// TwinCAT 3 PLC project SRC
// ProgramVersion: 3.1.4023.0
// libraries:
//   Tc2_Standard, * (Beckhoff Automation GmbH)
//   Tc2_System, * (Beckhoff Automation GmbH)
//   Tc3_JsonXml, * (Beckhoff Automation GmbH)
//   Tc3_Module, * (Beckhoff Automation GmbH)
// project tree:
//   DUTs/ENUM/ eCellState.TcDUT, eState.TcDUT
//   DUTs/STRUCT/HandledIO/Inputs/ st_IO_Inputs.TcDUT, st_PressureTransducer_Input.TcDUT, st_Robot_Input.TcDUT
//   DUTs/STRUCT/HandledIO/Outputs/ st_IO_Outputs.TcDUT, st_Pump_Output.TcDUT, st_Robot_Output.TcDUT
//   DUTs/STRUCT/Config/ ST_Configuration.TcDUT
//   DUTs/STRUCT/HMI/inputs/ st_PLCtoHMI_VariantControl.TcDUT, st_PLCtoHMI.TcDUT, st_PLCtoHMI_Hydrualics.TcDUT, st_PLCtoHMI_Cell.TcDUT, st_PLCtoHMI_PressureTrans.TcDUT, st_PLCtoHMI_Pump.TcDUT, st_PLCtoHMI_Robot.TcDUT
//   DUTs/STRUCT/HMI/outputs/ st_HMItoPLC.TcDUT, st_HMItoPLC_Cell.TcDUT, st_HMItoPLC_HMI.TcDUT, st_HMItoPLC_VariantControl.TcDUT
//   DUTs/STRUCT/IO/Base/ EtcMasterBase_62654B43.TcDUT, EtcSlaveBase_82538BE2.TcDUT, EtcSlaveBoxBase_77A0E4A7.TcDUT, EtcSlaveEndTerminalBase_866C7F0C.TcDUT, EtcSlaveTerminalBase_947E5A46.TcDUT, InputBase_8311D824.TcDUT, OutputBase_10CEE7DE.TcDUT, SyncUnitsBase_AD6C35CE.TcDUT, SyncUnitTaskBase_FCD3CBF3.TcDUT, SyncUnitTasksBase_7C8711EB.TcDUT
//   DUTs/STRUCT/IO/Boxes/ EK1100_1FC0878B.TcDUT, EL2634_7B64371E.TcDUT, EL3024_C4269E32.TcDUT, KRC4_secondary_EL6695_4F43E7C3.TcDUT
//   DUTs/STRUCT/IO/Devices/ SyncUnits_67D36DDA.TcDUT, SyncUnitTasks_4BE01469.TcDUT, SyncUnitTask_AB2F5079.TcDUT
//   DUTs/STRUCT/IO/PdoEntries/ FSOE_8292E3BB.TcDUT, FSOE_892AE692.TcDUT, Status_F2CE6D91.TcDUT
//   DUTs/STRUCT/IO/PDOs/ AI_Standard_Channel_4A394481.TcDUT, Channel_42CA91F7.TcDUT, Compact_1DE69B90.TcDUT, InfoData_32EB74EA.TcDUT, InfoData_6F19DB2B.TcDUT, InfoData_8649EEEB.TcDUT, InfoData_90184F0C.TcDUT, InfoData_E68C61CD.TcDUT, Inputs_A65FACA4.TcDUT, Inputs_Bitf_43DA21F5.TcDUT, Module_1_Sync_Inputs_26A07CFD.TcDUT, Module_2_Safety_Data_Bitf_8_Byte_x_D7FC8792.TcDUT, Module_3_Default_IO_1C907BA3.TcDUT, Outputs_23C0ED1D.TcDUT, Outputs_Bitf_2744F336.TcDUT, Std_In_4_Bytes_89628F68.TcDUT, Std_Out_4_Bytes_1F5BD6B7.TcDUT, WcState_0B2B16F9.TcDUT, WcState_9091E0EB.TcDUT
//   DUTs/STRUCT/IO/Topology/ E_Bus_F0495AE1.TcDUT, Term_1_EK1100_53501D32.TcDUT
//   / PlcTask.TcTTO
//   POUs/Cell/BaseClasses/ StateMachineBase.TcPOU
//   POUs/Cell/ FB_Cell.TcPOU
//   POUs/Cell/Hardware_IO/ FB_Topology.TcPOU
//   POUs/Cell/Hydrualics/ FB_HydrualicSystem.TcPOU
//   POUs/Cell/Hydrualics/PressureSensor/ FB_PressureSensor.TcPOU
//   POUs/Cell/Hydrualics/PressureSensor/Types/ FB_GenericBrand_Transceiver.TcPOU, FB_PressureTransceiver_Sim.TcPOU
//   POUs/Cell/Hydrualics/Pump/ FB_Pump.TcPOU
//   POUs/Cell/Hydrualics/Pump/Types/ FB_Pump_HPU.TcPOU, FB_Pump_RelayOnly.TcPOU, FB_Pump_Simulator.TcPOU
//   POUs/Cell/Robots/6_axis/Types/ FB_Fanuc.TcPOU, FB_Kuka_KRC2.TcPOU, FB_Kuka_KRC4.TcPOU, FB_Robot_Simulator.TcPOU
//   POUs/Cell/Robots/ FB_Robot.TcPOU
//   POUs/Cell/Robots/Gantry/Types/ FB_SomeGrantryRobot.TcPOU
//   POUs/Cell/_Interface/ I_HydrualicPump.TcIO, I_PressureSensor.TcIO, I_Robot.TcIO
//   POUs/ FB_VariantControl.TcPOU, MAIN.TcPOU
//   POUs/Functions/ Queue_FIFO.TcPOU, Scale.TcPOU
//   POUs/HMI/ FB_HMI.TcPOU
//   GVLs/ GVL_iXlinker.TcGVL

CONFIGURATION SRC
    RESOURCE PLC ON TwinCAT3
        TASK PlcTask(INTERVAL := T#10ms, PRIORITY := 20);
        PROGRAM MAIN WITH PlcTask : MAIN;
    END_RESOURCE
END_CONFIGURATION

// ---- DUTs/ENUM/eCellState.TcDUT
TYPE eCellState :
(
	eCellState_Manual, eCellState_Automatic, eCellState_Error
);
END_TYPE

// ---- DUTs/ENUM/eState.TcDUT
{attribute 'strict'}
{attribute 'to_string'}
TYPE eState :
(
	eState_Idle, eState_Startup, eState_Ready, eState_Running, eState_Complete, eState_Holding,
	eState_Held, eState_Stopping, eState_Stopped, eState_Error, eState_Independent, eState_Resetting, eState_Restarting,
	eState_Warmup
);
END_TYPE

// ---- DUTs/STRUCT/HandledIO/Inputs/st_IO_Inputs.TcDUT
TYPE st_IO_Inputs :
STRUCT
    robot :ST_Robot_Input;
    pressureTransducer : ST_PressureTransducer_Input;
END_STRUCT
END_TYPE

// ---- DUTs/STRUCT/HandledIO/Inputs/st_PressureTransducer_Input.TcDUT
TYPE st_PressureTransducer_Input :
STRUCT
	value : LREAL;
END_STRUCT
END_TYPE

// ---- DUTs/STRUCT/HandledIO/Inputs/st_Robot_Input.TcDUT
TYPE st_Robot_Input :
STRUCT
    fault : BOOL;
END_STRUCT
END_TYPE

// ---- DUTs/STRUCT/HandledIO/Outputs/st_IO_Outputs.TcDUT
TYPE st_IO_Outputs :
STRUCT
    hydroPump : ST_Pump_Output;
    robot : ST_Robot_Output;
END_STRUCT
END_TYPE

// ---- DUTs/STRUCT/HandledIO/Outputs/st_Pump_Output.TcDUT
TYPE st_Pump_Output :
STRUCT
	On : BOOL;
END_STRUCT
END_TYPE

// ---- DUTs/STRUCT/HandledIO/Outputs/st_Robot_Output.TcDUT
TYPE st_Robot_Output :
STRUCT
    fault : BOOL;
END_STRUCT
END_TYPE

// ---- DUTs/STRUCT/Config/ST_Configuration.TcDUT
TYPE ST_Configuration :
STRUCT
	sVersionHW : STRING;
	sVersionSW : STRING;

	// Which variant is active
	bIsV1_0_0 		: BOOL;
	bIsSimulator 	: BOOL;

	// Hydrualic pump definition
	bHasPump : BOOL;
	sPumpType : STRING;
	
	// Pressure sensor definition
	bHasPressureSensor : BOOL;
	sPressureSensorType : STRING;
    
    // Robot definition
    bHasRobot : BOOL;
    sRobotType : STRING;
END_STRUCT
END_TYPE

// ---- DUTs/STRUCT/HMI/inputs/st_PLCtoHMI_VariantControl.TcDUT
TYPE st_PLCtoHMI_VariantControl :
STRUCT
    bNeedsCellDefinition : BOOL;
END_STRUCT
END_TYPE

// ---- DUTs/STRUCT/HMI/inputs/st_PLCtoHMI.TcDUT
TYPE st_PLCtoHMI :
STRUCT
    cell : st_PLCtoHMI_Cell;
    robot : st_PLCtoHMI_Robot;
    hydrualics : st_PLCtoHMI_Hydrualics;
    variantControl : st_PLCtoHMI_VariantControl;
    //hmi : st_PLCtoHMI_HMI;
END_STRUCT
END_TYPE

// ---- DUTs/STRUCT/HMI/inputs/st_PLCtoHMI_Hydrualics.TcDUT
TYPE st_PLCtoHMI_Hydrualics :
STRUCT
    state : eState;
    psiSensor : st_PLCtoHMI_PressureTrans;
    pump : st_PLCtoHMI_Pump;
END_STRUCT
END_TYPE

// ---- DUTs/STRUCT/HMI/inputs/st_PLCtoHMI_Cell.TcDUT
TYPE st_PLCtoHMI_Cell :
STRUCT
    state : eCellState;
    bPower : BOOL; // power hydrualics maybe?
    bGoToManual: BOOL;
	bGoToAuto: BOOL;
	bReset : BOOL;
END_STRUCT
END_TYPE

// ---- DUTs/STRUCT/HMI/inputs/st_PLCtoHMI_PressureTrans.TcDUT
TYPE st_PLCtoHMI_PressureTrans :
STRUCT
    value : LREAL;
END_STRUCT
END_TYPE

// ---- DUTs/STRUCT/HMI/inputs/st_PLCtoHMI_Pump.TcDUT
TYPE st_PLCtoHMI_Pump :
STRUCT
    state : eState;
END_STRUCT
END_TYPE

// ---- DUTs/STRUCT/HMI/inputs/st_PLCtoHMI_Robot.TcDUT
TYPE st_PLCtoHMI_Robot :
STRUCT
    state : eState;
END_STRUCT
END_TYPE

// ---- DUTs/STRUCT/HMI/outputs/st_HMItoPLC.TcDUT
TYPE st_HMItoPLC :
STRUCT
    cell : st_HMItoPLC_Cell;
    hmi : st_HMItoPLC_HMI;
    variantControl : st_HMItoPLC_VariantControl;
END_STRUCT
END_TYPE

// ---- DUTs/STRUCT/HMI/outputs/st_HMItoPLC_Cell.TcDUT
TYPE st_HMItoPLC_Cell :
STRUCT
    bPower : BOOL; // power hydrualics maybe?
    bGoToManual: BOOL;
	bGoToAuto: BOOL;
	bReset : BOOL;
END_STRUCT
END_TYPE

// ---- DUTs/STRUCT/HMI/outputs/st_HMItoPLC_HMI.TcDUT
TYPE st_HMItoPLC_HMI :
STRUCT
    bAutoManual_btn : BOOL;
    bShowResetBtn : BOOL;
END_STRUCT
END_TYPE

// ---- DUTs/STRUCT/HMI/outputs/st_HMItoPLC_VariantControl.TcDUT
TYPE st_HMItoPLC_VariantControl :
STRUCT
    bExportJSON : BOOL;
    bWriteJSON : BOOL;
    Config : ST_Configuration;
    bNeedsCellDefinition : BOOL;
END_STRUCT
END_TYPE

// ---- DUTs/STRUCT/IO/Base/EtcMasterBase_62654B43.TcDUT

TYPE EtcMasterBase_62654B43 :
STRUCT
END_STRUCT
END_TYPE

// ---- DUTs/STRUCT/IO/Base/EtcSlaveBase_82538BE2.TcDUT

TYPE EtcSlaveBase_82538BE2 :
STRUCT
END_STRUCT
END_TYPE

// ---- DUTs/STRUCT/IO/Base/EtcSlaveBoxBase_77A0E4A7.TcDUT

{attribute clr[Container(Layout.Stack)]}
{attribute clr[Group(Layout.GroupBox)]}
{attribute addProperty PreviousPort "Unknown"}
{attribute addProperty SyncUnit "Unknown"}
TYPE EtcSlaveBoxBase_77A0E4A7 EXTENDS EtcSlaveBase_82538BE2 :
STRUCT
END_STRUCT
END_TYPE

// ---- DUTs/STRUCT/IO/Base/EtcSlaveEndTerminalBase_866C7F0C.TcDUT

{attribute clr[Container(Layout.Stack)]}
{attribute clr[Group(Layout.GroupBox)]}
{attribute addProperty PreviousPort "Unknown"}
{attribute addProperty SyncUnit "Unknown"}
TYPE EtcSlaveEndTerminalBase_866C7F0C EXTENDS EtcSlaveBase_82538BE2 :
STRUCT
END_STRUCT
END_TYPE

// ---- DUTs/STRUCT/IO/Base/EtcSlaveTerminalBase_947E5A46.TcDUT

{attribute clr[Container(Layout.Stack)]}
{attribute clr[Group(Layout.GroupBox)]}
{attribute addProperty PreviousPort "Unknown"}
{attribute addProperty SyncUnit "Unknown"}
TYPE EtcSlaveTerminalBase_947E5A46 EXTENDS EtcSlaveBase_82538BE2 :
STRUCT
END_STRUCT
END_TYPE

// ---- DUTs/STRUCT/IO/Base/InputBase_8311D824.TcDUT

TYPE InputBase_8311D824 :
STRUCT
END_STRUCT
END_TYPE

// ---- DUTs/STRUCT/IO/Base/OutputBase_10CEE7DE.TcDUT

TYPE OutputBase_10CEE7DE :
STRUCT
END_STRUCT
END_TYPE

// ---- DUTs/STRUCT/IO/Base/SyncUnitsBase_AD6C35CE.TcDUT

TYPE SyncUnitsBase_AD6C35CE :
STRUCT
END_STRUCT
END_TYPE

// ---- DUTs/STRUCT/IO/Base/SyncUnitTaskBase_FCD3CBF3.TcDUT

TYPE SyncUnitTaskBase_FCD3CBF3 :
STRUCT
END_STRUCT
END_TYPE

// ---- DUTs/STRUCT/IO/Base/SyncUnitTasksBase_7C8711EB.TcDUT

TYPE SyncUnitTasksBase_7C8711EB :
STRUCT
END_STRUCT
END_TYPE

// ---- DUTs/STRUCT/IO/Boxes/EK1100_1FC0878B.TcDUT
{attribute 'GeneratedUsingTerminal: EK1100-0000-0018'}
{attribute addProperty VendorId "#x00000002"}
{attribute addProperty BoxType "EK1100-0000-0018"}
{attribute addProperty Description "EK1100 EtherCAT Coupler (2A E-Bus)"}
{attribute addProperty Physics "YKY"}
{attribute addProperty Id "InfoDataAT %I*InfoData_6F19DB2B2"}
{attribute addProperty CRC "532711307"}
{attribute addProperty Size "2"}
TYPE EK1100_1FC0878B EXTENDS EtcSlaveBoxBase_77A0E4A7 :
STRUCT
	{attribute addProperty Name "InfoData"}
	InfoData : InfoData_6F19DB2B;
END_STRUCT
END_TYPE

// ---- DUTs/STRUCT/IO/Boxes/EL2634_7B64371E.TcDUT
{attribute 'GeneratedUsingTerminal: EL2634-0000-0017'}
{attribute addProperty VendorId "#x00000002"}
{attribute addProperty BoxType "EL2634-0000-0017"}
{attribute addProperty Description "EL2634 4Ch. Relay Output, NO (250V AC / 30V DC)"}
{attribute addProperty Physics "KK"}
{attribute addProperty Id "Channel_1AT %Q*Channel_42CA91F71Channel_2AT %Q*Channel_42CA91F71Channel_3AT %Q*Channel_42CA91F71Channel_4AT %Q*Channel_42CA91F71WcStateAT %I*WcState_0B2B16F91InfoDataAT %I*InfoData_6F19DB2B2"}
{attribute addProperty CRC "2070165278"}
{attribute addProperty Size "7"}
TYPE EL2634_7B64371E EXTENDS EtcSlaveTerminalBase_947E5A46 :
STRUCT
	{attribute addProperty Name "Channel_1"}
	Channel_1 : Channel_42CA91F7;
	{attribute addProperty Name "Channel_2"}
	Channel_2 : Channel_42CA91F7;
	{attribute addProperty Name "Channel_3"}
	Channel_3 : Channel_42CA91F7;
	{attribute addProperty Name "Channel_4"}
	Channel_4 : Channel_42CA91F7;
	{attribute addProperty Name "WcState"}
	WcState : WcState_0B2B16F9;
	{attribute addProperty Name "InfoData"}
	InfoData : InfoData_6F19DB2B;
END_STRUCT
END_TYPE

// ---- DUTs/STRUCT/IO/Boxes/EL3024_C4269E32.TcDUT
{attribute 'GeneratedUsingTerminal: EL3024-0000-0019'}
{attribute addProperty VendorId "#x00000002"}
{attribute addProperty BoxType "EL3024-0000-0019"}
{attribute addProperty Description "EL3024 4Ch. Ana. Input 4-20mA DIFF"}
{attribute addProperty Physics "KK"}
{attribute addProperty Id "AI_Standard_Channel_1AT %I*AI_Standard_Channel_4A3944819AI_Standard_Channel_2AT %I*AI_Standard_Channel_4A3944819AI_Standard_Channel_3AT %I*AI_Standard_Channel_4A3944819AI_Standard_Channel_4AT %I*AI_Standard_Channel_4A3944819WcStateAT %I*WcState_9091E0EB2InfoDataAT %I*InfoData_32EB74EA10"}
{attribute addProperty CRC "3290865202"}
{attribute addProperty Size "48"}
TYPE EL3024_C4269E32 EXTENDS EtcSlaveTerminalBase_947E5A46 :
STRUCT
	{attribute addProperty Name "AI_Standard_Channel_1"}
	AI_Standard_Channel_1 : AI_Standard_Channel_4A394481;
	{attribute addProperty Name "AI_Standard_Channel_2"}
	AI_Standard_Channel_2 : AI_Standard_Channel_4A394481;
	{attribute addProperty Name "AI_Standard_Channel_3"}
	AI_Standard_Channel_3 : AI_Standard_Channel_4A394481;
	{attribute addProperty Name "AI_Standard_Channel_4"}
	AI_Standard_Channel_4 : AI_Standard_Channel_4A394481;
	{attribute addProperty Name "WcState"}
	WcState : WcState_9091E0EB;
	{attribute addProperty Name "InfoData"}
	InfoData : InfoData_32EB74EA;
END_STRUCT
END_TYPE

// ---- DUTs/STRUCT/IO/Boxes/KRC4_secondary_EL6695_4F43E7C3.TcDUT
{attribute 'GeneratedUsingTerminal: KRC4 secondary EL6695-1001-0004'}
{attribute addProperty VendorId "#x000060c8"}
{attribute addProperty BoxType "KRC4 secondary EL6695-1001-0004"}
{attribute addProperty Description "KRC4 secondary EL6695-1001"}
{attribute addProperty Physics "YY"}
{attribute addProperty Id "Module_1_Sync_InputsModule_1_Sync_Inputs_26A07CFD3Module_2_Safety_Data_Bitf_8_Byte_xModule_2_Safety_Data_Bitf_8_Byte_x_D7FC8792150Module_3_Default_IOModule_3_Default_IO_1C907BA38WcStateAT %I*WcState_9091E0EB2InfoDataAT %I*InfoData_90184F0C16"}
{attribute addProperty CRC "1329850307"}
{attribute addProperty Size "179"}
TYPE KRC4_secondary_EL6695_4F43E7C3 EXTENDS EtcSlaveBoxBase_77A0E4A7 :
STRUCT
	{attribute addProperty Name "Module_1_Sync_Inputs"}
	Module_1_Sync_Inputs : Module_1_Sync_Inputs_26A07CFD;
	{attribute addProperty Name "Module_2_Safety_Data_Bitf_8_Byte_x"}
	Module_2_Safety_Data_Bitf_8_Byte_x : Module_2_Safety_Data_Bitf_8_Byte_x_D7FC8792;
	{attribute addProperty Name "Module_3_Default_IO"}
	Module_3_Default_IO : Module_3_Default_IO_1C907BA3;
	{attribute addProperty Name "WcState"}
	WcState : WcState_9091E0EB;
	{attribute addProperty Name "InfoData"}
	InfoData : InfoData_90184F0C;
END_STRUCT
END_TYPE

// ---- DUTs/STRUCT/IO/Devices/SyncUnits_67D36DDA.TcDUT
{attribute 'GeneratedUsingTerminal: '}
{attribute addProperty BoxType ""}
{attribute addProperty Id "_defaultAT %I*SyncUnitTasks_4BE0146918"}
{attribute addProperty CRC "1741909466"}
{attribute addProperty Size "18"}
TYPE SyncUnits_67D36DDA EXTENDS SyncUnitsBase_AD6C35CE :
STRUCT
	{attribute addProperty Name "_default"}
	_default : SyncUnitTasks_4BE01469;
END_STRUCT
END_TYPE

// ---- DUTs/STRUCT/IO/Devices/SyncUnitTasks_4BE01469.TcDUT
{attribute 'GeneratedUsingTerminal: '}
{attribute addProperty BoxType ""}
{attribute addProperty Id "unreferencedAT %I*SyncUnitTask_AB2F50799PlcTaskAT %I*SyncUnitTask_AB2F50799"}
{attribute addProperty CRC "1272976489"}
{attribute addProperty Size "18"}
TYPE SyncUnitTasks_4BE01469 EXTENDS SyncUnitTasksBase_7C8711EB :
STRUCT
	{attribute addProperty Name "unreferenced"}
	unreferenced : SyncUnitTask_AB2F5079;
	{attribute addProperty Name "PlcTask"}
	PlcTask : SyncUnitTask_AB2F5079;
END_STRUCT
END_TYPE

// ---- DUTs/STRUCT/IO/Devices/SyncUnitTask_AB2F5079.TcDUT
{attribute 'GeneratedUsingTerminal: IODEVICETYPE_ETHERCATPROT'}
{attribute addProperty BoxType "IODEVICETYPE_ETHERCATPROT"}
{attribute addProperty Id "WcStateAT %I*WcState_0B2B16F91InfoDataAT %I*InfoData_8649EEEB8"}
{attribute addProperty CRC "2872004729"}
{attribute addProperty Size "9"}
TYPE SyncUnitTask_AB2F5079 EXTENDS SyncUnitTaskBase_FCD3CBF3 :
STRUCT
	{attribute addProperty Name "WcState"}
	WcState : WcState_0B2B16F9;
	{attribute addProperty Name "InfoData"}
	InfoData : InfoData_8649EEEB;
END_STRUCT
END_TYPE

// ---- DUTs/STRUCT/IO/PdoEntries/FSOE_8292E3BB.TcDUT
{attribute 'GeneratedUsingTerminal: KRC4 secondary EL6695-1001-0004'}
{attribute addProperty BoxType "KRC4 secondary EL6695-1001-0004"}
{attribute addProperty Id "FSOE_CommandUSINT1FSOE_Out_D_0_RES_1BOOL1FSOE_Out_D_0_NHEBOOL1FSOE_Out_D_0_BSBOOL1FSOE_Out_D_0_QBSBOOL1FSOE_Out_D_0_SHS1BOOL1FSOE_Out_D_0_SHS2BOOL1FSOE_Out_D_0_E2BOOL1FSOE_Out_D_0_E7BOOL1FSOE_Out_D_0_US2BOOL1FSOE_Out_D_0_SBHBOOL1FSOE_Out_D_0_RES_4BOOL1FSOE_Out_D_0_RES_5BOOL1FSOE_Out_D_0_RES_6BOOL1FSOE_Out_D_0_RES_7BOOL1FSOE_Out_D_0_RES_8BOOL1FSOE_Out_D_0_SPABOOL1FSOE_Master_CRC_0UINT2FSOE_Out_D_1_JRBOOL1FSOE_Out_D_1_VREDBOOL1FSOE_Out_D_1_SBH_1BOOL1FSOE_Out_D_1_SBH_2BOOL1FSOE_Out_D_1_SBH_3BOOL1FSOE_Out_D_1_SBH_4BOOL1FSOE_Out_D_1_SBH_5BOOL1FSOE_Out_D_1_SBH_6BOOL1FSOE_Out_D_1_RES_1BOOL1FSOE_Out_D_1_RES_2BOOL1FSOE_Out_D_1_RES_3BOOL1FSOE_Out_D_1_RES_4BOOL1FSOE_Out_D_1_RES_5BOOL1FSOE_Out_D_1_RES_6BOOL1FSOE_Out_D_1_RES_7BOOL1FSOE_Out_D_1_RES_8BOOL1FSOE_Master_CRC_1UINT2FSOE_Out_D_2_UER1BOOL1FSOE_Out_D_2_UER2BOOL1FSOE_Out_D_2_UER3BOOL1FSOE_Out_D_2_UER4BOOL1FSOE_Out_D_2_UER5BOOL1FSOE_Out_D_2_UER6BOOL1FSOE_Out_D_2_UER7BOOL1FSOE_Out_D_2_UER8BOOL1FSOE_Out_D_2_UER9BOOL1FSOE_Out_D_2_UER10BOOL1FSOE_Out_D_2_UER11BOOL1FSOE_Out_D_2_UER12BOOL1FSOE_Out_D_2_UER13BOOL1FSOE_Out_D_2_UER14BOOL1FSOE_Out_D_2_UER15BOOL1FSOE_Out_D_2_UER16BOOL1FSOE_Master_CRC_2UINT2FSOE_Out_D_3_WZ1BOOL1FSOE_Out_D_3_WZ2BOOL1FSOE_Out_D_3_WZ3BOOL1FSOE_Out_D_3_WZ4BOOL1FSOE_Out_D_3_WZ5BOOL1FSOE_Out_D_3_WZ6BOOL1FSOE_Out_D_3_WZ7BOOL1FSOE_Out_D_3_WZ8BOOL1FSOE_Out_D_3_WZ9BOOL1FSOE_Out_D_3_WZ10BOOL1FSOE_Out_D_3_WZ11BOOL1FSOE_Out_D_3_WZ12BOOL1FSOE_Out_D_3_WZ13BOOL1FSOE_Out_D_3_WZ14BOOL1FSOE_Out_D_3_WZ15BOOL1FSOE_Out_D_3_WZ16BOOL1FSOE_Master_CRC_3UINT2FSOE_ConnIDUINT2"}
{attribute addProperty CRC "2190664635"}
{attribute addProperty Size "75"}
TYPE FSOE_8292E3BB :
STRUCT
	{attribute addProperty Name "FSOE_Command"}
	FSOE_Command : USINT;
	{attribute addProperty Name "FSOE_Out_D_0_RES_1"}
	FSOE_Out_D_0_RES_1 : BOOL;
	{attribute addProperty Name "FSOE_Out_D_0_NHE"}
	FSOE_Out_D_0_NHE : BOOL;
	{attribute addProperty Name "FSOE_Out_D_0_BS"}
	FSOE_Out_D_0_BS : BOOL;
	{attribute addProperty Name "FSOE_Out_D_0_QBS"}
	FSOE_Out_D_0_QBS : BOOL;
	{attribute addProperty Name "FSOE_Out_D_0_SHS1"}
	FSOE_Out_D_0_SHS1 : BOOL;
	{attribute addProperty Name "FSOE_Out_D_0_SHS2"}
	FSOE_Out_D_0_SHS2 : BOOL;
	{attribute addProperty Name "FSOE_Out_D_0_E2"}
	FSOE_Out_D_0_E2 : BOOL;
	{attribute addProperty Name "FSOE_Out_D_0_E7"}
	FSOE_Out_D_0_E7 : BOOL;
	{attribute addProperty Name "FSOE_Out_D_0_US2"}
	FSOE_Out_D_0_US2 : BOOL;
	{attribute addProperty Name "FSOE_Out_D_0_SBH"}
	FSOE_Out_D_0_SBH : BOOL;
	{attribute addProperty Name "FSOE_Out_D_0_RES_4"}
	FSOE_Out_D_0_RES_4 : BOOL;
	{attribute addProperty Name "FSOE_Out_D_0_RES_5"}
	FSOE_Out_D_0_RES_5 : BOOL;
	{attribute addProperty Name "FSOE_Out_D_0_RES_6"}
	FSOE_Out_D_0_RES_6 : BOOL;
	{attribute addProperty Name "FSOE_Out_D_0_RES_7"}
	FSOE_Out_D_0_RES_7 : BOOL;
	{attribute addProperty Name "FSOE_Out_D_0_RES_8"}
	FSOE_Out_D_0_RES_8 : BOOL;
	{attribute addProperty Name "FSOE_Out_D_0_SPA"}
	FSOE_Out_D_0_SPA : BOOL;
	{attribute addProperty Name "FSOE_Master_CRC_0"}
	FSOE_Master_CRC_0 : UINT;
	{attribute addProperty Name "FSOE_Out_D_1_JR"}
	FSOE_Out_D_1_JR : BOOL;
	{attribute addProperty Name "FSOE_Out_D_1_VRED"}
	FSOE_Out_D_1_VRED : BOOL;
	{attribute addProperty Name "FSOE_Out_D_1_SBH_1"}
	FSOE_Out_D_1_SBH_1 : BOOL;
	{attribute addProperty Name "FSOE_Out_D_1_SBH_2"}
	FSOE_Out_D_1_SBH_2 : BOOL;
	{attribute addProperty Name "FSOE_Out_D_1_SBH_3"}
	FSOE_Out_D_1_SBH_3 : BOOL;
	{attribute addProperty Name "FSOE_Out_D_1_SBH_4"}
	FSOE_Out_D_1_SBH_4 : BOOL;
	{attribute addProperty Name "FSOE_Out_D_1_SBH_5"}
	FSOE_Out_D_1_SBH_5 : BOOL;
	{attribute addProperty Name "FSOE_Out_D_1_SBH_6"}
	FSOE_Out_D_1_SBH_6 : BOOL;
	{attribute addProperty Name "FSOE_Out_D_1_RES_1"}
	FSOE_Out_D_1_RES_1 : BOOL;
	{attribute addProperty Name "FSOE_Out_D_1_RES_2"}
	FSOE_Out_D_1_RES_2 : BOOL;
	{attribute addProperty Name "FSOE_Out_D_1_RES_3"}
	FSOE_Out_D_1_RES_3 : BOOL;
	{attribute addProperty Name "FSOE_Out_D_1_RES_4"}
	FSOE_Out_D_1_RES_4 : BOOL;
	{attribute addProperty Name "FSOE_Out_D_1_RES_5"}
	FSOE_Out_D_1_RES_5 : BOOL;
	{attribute addProperty Name "FSOE_Out_D_1_RES_6"}
	FSOE_Out_D_1_RES_6 : BOOL;
	{attribute addProperty Name "FSOE_Out_D_1_RES_7"}
	FSOE_Out_D_1_RES_7 : BOOL;
	{attribute addProperty Name "FSOE_Out_D_1_RES_8"}
	FSOE_Out_D_1_RES_8 : BOOL;
	{attribute addProperty Name "FSOE_Master_CRC_1"}
	FSOE_Master_CRC_1 : UINT;
	{attribute addProperty Name "FSOE_Out_D_2_UER1"}
	FSOE_Out_D_2_UER1 : BOOL;
	{attribute addProperty Name "FSOE_Out_D_2_UER2"}
	FSOE_Out_D_2_UER2 : BOOL;
	{attribute addProperty Name "FSOE_Out_D_2_UER3"}
	FSOE_Out_D_2_UER3 : BOOL;
	{attribute addProperty Name "FSOE_Out_D_2_UER4"}
	FSOE_Out_D_2_UER4 : BOOL;
	{attribute addProperty Name "FSOE_Out_D_2_UER5"}
	FSOE_Out_D_2_UER5 : BOOL;
	{attribute addProperty Name "FSOE_Out_D_2_UER6"}
	FSOE_Out_D_2_UER6 : BOOL;
	{attribute addProperty Name "FSOE_Out_D_2_UER7"}
	FSOE_Out_D_2_UER7 : BOOL;
	{attribute addProperty Name "FSOE_Out_D_2_UER8"}
	FSOE_Out_D_2_UER8 : BOOL;
	{attribute addProperty Name "FSOE_Out_D_2_UER9"}
	FSOE_Out_D_2_UER9 : BOOL;
	{attribute addProperty Name "FSOE_Out_D_2_UER10"}
	FSOE_Out_D_2_UER10 : BOOL;
	{attribute addProperty Name "FSOE_Out_D_2_UER11"}
	FSOE_Out_D_2_UER11 : BOOL;
	{attribute addProperty Name "FSOE_Out_D_2_UER12"}
	FSOE_Out_D_2_UER12 : BOOL;
	{attribute addProperty Name "FSOE_Out_D_2_UER13"}
	FSOE_Out_D_2_UER13 : BOOL;
	{attribute addProperty Name "FSOE_Out_D_2_UER14"}
	FSOE_Out_D_2_UER14 : BOOL;
	{attribute addProperty Name "FSOE_Out_D_2_UER15"}
	FSOE_Out_D_2_UER15 : BOOL;
	{attribute addProperty Name "FSOE_Out_D_2_UER16"}
	FSOE_Out_D_2_UER16 : BOOL;
	{attribute addProperty Name "FSOE_Master_CRC_2"}
	FSOE_Master_CRC_2 : UINT;
	{attribute addProperty Name "FSOE_Out_D_3_WZ1"}
	FSOE_Out_D_3_WZ1 : BOOL;
	{attribute addProperty Name "FSOE_Out_D_3_WZ2"}
	FSOE_Out_D_3_WZ2 : BOOL;
	{attribute addProperty Name "FSOE_Out_D_3_WZ3"}
	FSOE_Out_D_3_WZ3 : BOOL;
	{attribute addProperty Name "FSOE_Out_D_3_WZ4"}
	FSOE_Out_D_3_WZ4 : BOOL;
	{attribute addProperty Name "FSOE_Out_D_3_WZ5"}
	FSOE_Out_D_3_WZ5 : BOOL;
	{attribute addProperty Name "FSOE_Out_D_3_WZ6"}
	FSOE_Out_D_3_WZ6 : BOOL;
	{attribute addProperty Name "FSOE_Out_D_3_WZ7"}
	FSOE_Out_D_3_WZ7 : BOOL;
	{attribute addProperty Name "FSOE_Out_D_3_WZ8"}
	FSOE_Out_D_3_WZ8 : BOOL;
	{attribute addProperty Name "FSOE_Out_D_3_WZ9"}
	FSOE_Out_D_3_WZ9 : BOOL;
	{attribute addProperty Name "FSOE_Out_D_3_WZ10"}
	FSOE_Out_D_3_WZ10 : BOOL;
	{attribute addProperty Name "FSOE_Out_D_3_WZ11"}
	FSOE_Out_D_3_WZ11 : BOOL;
	{attribute addProperty Name "FSOE_Out_D_3_WZ12"}
	FSOE_Out_D_3_WZ12 : BOOL;
	{attribute addProperty Name "FSOE_Out_D_3_WZ13"}
	FSOE_Out_D_3_WZ13 : BOOL;
	{attribute addProperty Name "FSOE_Out_D_3_WZ14"}
	FSOE_Out_D_3_WZ14 : BOOL;
	{attribute addProperty Name "FSOE_Out_D_3_WZ15"}
	FSOE_Out_D_3_WZ15 : BOOL;
	{attribute addProperty Name "FSOE_Out_D_3_WZ16"}
	FSOE_Out_D_3_WZ16 : BOOL;
	{attribute addProperty Name "FSOE_Master_CRC_3"}
	FSOE_Master_CRC_3 : UINT;
	{attribute addProperty Name "FSOE_ConnID"}
	FSOE_ConnID : UINT;
END_STRUCT
END_TYPE

// ---- DUTs/STRUCT/IO/PdoEntries/FSOE_892AE692.TcDUT
{attribute 'GeneratedUsingTerminal: KRC4 secondary EL6695-1001-0004'}
{attribute addProperty BoxType "KRC4 secondary EL6695-1001-0004"}
{attribute addProperty Id "FSOE_CommandUSINT1FSOE_Inp_D_0_NHLBOOL1FSOE_Inp_D_0_AFBOOL1FSOE_Inp_D_0_FFBOOL1FSOE_Inp_D_0_ZSBOOL1FSOE_Inp_D_0_PEBOOL1FSOE_Inp_D_0_EXTBOOL1FSOE_Inp_D_0_T1BOOL1FSOE_Inp_D_0_T2BOOL1FSOE_Inp_D_0_NHEBOOL1FSOE_Inp_D_0_BSQBOOL1FSOE_Inp_D_0_SHS1BOOL1FSOE_Inp_D_0_SHS2BOOL1FSOE_Inp_D_0_RES_13BOOL1FSOE_Inp_D_0_RES_14BOOL1FSOE_Inp_D_0_PSABOOL1FSOE_Inp_D_0_SPBOOL1FSOE_Slave_CRC_0UINT2FSOE_Inp_D_1_SOBOOL1FSOE_Inp_D_1_RRBOOL1FSOE_Inp_D_1_JFBOOL1FSOE_Inp_D_1_VREDBOOL1FSOE_Inp_D_1_SBH_1BOOL1FSOE_Inp_D_1_SBH_2BOOL1FSOE_Inp_D_1_SBH_3BOOL1FSOE_Inp_D_1_SBH_4BOOL1FSOE_Inp_D_1_SBH_5BOOL1FSOE_Inp_D_1_SBH_6BOOL1FSOE_Inp_D_1_SOSBOOL1FSOE_Inp_D_1_RES_28BOOL1FSOE_Inp_D_1_RES_29BOOL1FSOE_Inp_D_1_RES_30BOOL1FSOE_Inp_D_1_RES_31BOOL1FSOE_Inp_D_1_RES_32BOOL1FSOE_Slave_CRC_1UINT2FSOE_Inp_D_2_MR1BOOL1FSOE_Inp_D_2_MR2BOOL1FSOE_Inp_D_2_MR3BOOL1FSOE_Inp_D_2_MR4BOOL1FSOE_Inp_D_2_MR5BOOL1FSOE_Inp_D_2_MR6BOOL1FSOE_Inp_D_2_MR7BOOL1FSOE_Inp_D_2_MR8BOOL1FSOE_Inp_D_2_MR9BOOL1FSOE_Inp_D_2_MR10BOOL1FSOE_Inp_D_2_MR11BOOL1FSOE_Inp_D_2_MR12BOOL1FSOE_Inp_D_2_MR13BOOL1FSOE_Inp_D_2_MR14BOOL1FSOE_Inp_D_2_MR15BOOL1FSOE_Inp_D_2_MR16BOOL1FSOE_Slave_CRC_2UINT2FSOE_Inp_D_3_RES_49BOOL1FSOE_Inp_D_3_RES_50BOOL1FSOE_Inp_D_3_RES_51BOOL1FSOE_Inp_D_3_RES_52BOOL1FSOE_Inp_D_3_RES_53BOOL1FSOE_Inp_D_3_RES_54BOOL1FSOE_Inp_D_3_RES_55BOOL1FSOE_Inp_D_3_RES_56BOOL1FSOE_Inp_D_3_RES_57BOOL1FSOE_Inp_D_3_RES_58BOOL1FSOE_Inp_D_3_RES_59BOOL1FSOE_Inp_D_3_RES_60BOOL1FSOE_Inp_D_3_RES_61BOOL1FSOE_Inp_D_3_RES_62BOOL1FSOE_Inp_D_3_RES_63BOOL1FSOE_Inp_D_3_RES_64BOOL1FSOE_Slave_CRC_3UINT2FSOE_ConnIDUINT2"}
{attribute addProperty CRC "2301290130"}
{attribute addProperty Size "75"}
TYPE FSOE_892AE692 :
STRUCT
	{attribute addProperty Name "FSOE_Command"}
	FSOE_Command : USINT;
	{attribute addProperty Name "FSOE_Inp_D_0_NHL"}
	FSOE_Inp_D_0_NHL : BOOL;
	{attribute addProperty Name "FSOE_Inp_D_0_AF"}
	FSOE_Inp_D_0_AF : BOOL;
	{attribute addProperty Name "FSOE_Inp_D_0_FF"}
	FSOE_Inp_D_0_FF : BOOL;
	{attribute addProperty Name "FSOE_Inp_D_0_ZS"}
	FSOE_Inp_D_0_ZS : BOOL;
	{attribute addProperty Name "FSOE_Inp_D_0_PE"}
	FSOE_Inp_D_0_PE : BOOL;
	{attribute addProperty Name "FSOE_Inp_D_0_EXT"}
	FSOE_Inp_D_0_EXT : BOOL;
	{attribute addProperty Name "FSOE_Inp_D_0_T1"}
	FSOE_Inp_D_0_T1 : BOOL;
	{attribute addProperty Name "FSOE_Inp_D_0_T2"}
	FSOE_Inp_D_0_T2 : BOOL;
	{attribute addProperty Name "FSOE_Inp_D_0_NHE"}
	FSOE_Inp_D_0_NHE : BOOL;
	{attribute addProperty Name "FSOE_Inp_D_0_BSQ"}
	FSOE_Inp_D_0_BSQ : BOOL;
	{attribute addProperty Name "FSOE_Inp_D_0_SHS1"}
	FSOE_Inp_D_0_SHS1 : BOOL;
	{attribute addProperty Name "FSOE_Inp_D_0_SHS2"}
	FSOE_Inp_D_0_SHS2 : BOOL;
	{attribute addProperty Name "FSOE_Inp_D_0_RES_13"}
	FSOE_Inp_D_0_RES_13 : BOOL;
	{attribute addProperty Name "FSOE_Inp_D_0_RES_14"}
	FSOE_Inp_D_0_RES_14 : BOOL;
	{attribute addProperty Name "FSOE_Inp_D_0_PSA"}
	FSOE_Inp_D_0_PSA : BOOL;
	{attribute addProperty Name "FSOE_Inp_D_0_SP"}
	FSOE_Inp_D_0_SP : BOOL;
	{attribute addProperty Name "FSOE_Slave_CRC_0"}
	FSOE_Slave_CRC_0 : UINT;
	{attribute addProperty Name "FSOE_Inp_D_1_SO"}
	FSOE_Inp_D_1_SO : BOOL;
	{attribute addProperty Name "FSOE_Inp_D_1_RR"}
	FSOE_Inp_D_1_RR : BOOL;
	{attribute addProperty Name "FSOE_Inp_D_1_JF"}
	FSOE_Inp_D_1_JF : BOOL;
	{attribute addProperty Name "FSOE_Inp_D_1_VRED"}
	FSOE_Inp_D_1_VRED : BOOL;
	{attribute addProperty Name "FSOE_Inp_D_1_SBH_1"}
	FSOE_Inp_D_1_SBH_1 : BOOL;
	{attribute addProperty Name "FSOE_Inp_D_1_SBH_2"}
	FSOE_Inp_D_1_SBH_2 : BOOL;
	{attribute addProperty Name "FSOE_Inp_D_1_SBH_3"}
	FSOE_Inp_D_1_SBH_3 : BOOL;
	{attribute addProperty Name "FSOE_Inp_D_1_SBH_4"}
	FSOE_Inp_D_1_SBH_4 : BOOL;
	{attribute addProperty Name "FSOE_Inp_D_1_SBH_5"}
	FSOE_Inp_D_1_SBH_5 : BOOL;
	{attribute addProperty Name "FSOE_Inp_D_1_SBH_6"}
	FSOE_Inp_D_1_SBH_6 : BOOL;
	{attribute addProperty Name "FSOE_Inp_D_1_SOS"}
	FSOE_Inp_D_1_SOS : BOOL;
	{attribute addProperty Name "FSOE_Inp_D_1_RES_28"}
	FSOE_Inp_D_1_RES_28 : BOOL;
	{attribute addProperty Name "FSOE_Inp_D_1_RES_29"}
	FSOE_Inp_D_1_RES_29 : BOOL;
	{attribute addProperty Name "FSOE_Inp_D_1_RES_30"}
	FSOE_Inp_D_1_RES_30 : BOOL;
	{attribute addProperty Name "FSOE_Inp_D_1_RES_31"}
	FSOE_Inp_D_1_RES_31 : BOOL;
	{attribute addProperty Name "FSOE_Inp_D_1_RES_32"}
	FSOE_Inp_D_1_RES_32 : BOOL;
	{attribute addProperty Name "FSOE_Slave_CRC_1"}
	FSOE_Slave_CRC_1 : UINT;
	{attribute addProperty Name "FSOE_Inp_D_2_MR1"}
	FSOE_Inp_D_2_MR1 : BOOL;
	{attribute addProperty Name "FSOE_Inp_D_2_MR2"}
	FSOE_Inp_D_2_MR2 : BOOL;
	{attribute addProperty Name "FSOE_Inp_D_2_MR3"}
	FSOE_Inp_D_2_MR3 : BOOL;
	{attribute addProperty Name "FSOE_Inp_D_2_MR4"}
	FSOE_Inp_D_2_MR4 : BOOL;
	{attribute addProperty Name "FSOE_Inp_D_2_MR5"}
	FSOE_Inp_D_2_MR5 : BOOL;
	{attribute addProperty Name "FSOE_Inp_D_2_MR6"}
	FSOE_Inp_D_2_MR6 : BOOL;
	{attribute addProperty Name "FSOE_Inp_D_2_MR7"}
	FSOE_Inp_D_2_MR7 : BOOL;
	{attribute addProperty Name "FSOE_Inp_D_2_MR8"}
	FSOE_Inp_D_2_MR8 : BOOL;
	{attribute addProperty Name "FSOE_Inp_D_2_MR9"}
	FSOE_Inp_D_2_MR9 : BOOL;
	{attribute addProperty Name "FSOE_Inp_D_2_MR10"}
	FSOE_Inp_D_2_MR10 : BOOL;
	{attribute addProperty Name "FSOE_Inp_D_2_MR11"}
	FSOE_Inp_D_2_MR11 : BOOL;
	{attribute addProperty Name "FSOE_Inp_D_2_MR12"}
	FSOE_Inp_D_2_MR12 : BOOL;
	{attribute addProperty Name "FSOE_Inp_D_2_MR13"}
	FSOE_Inp_D_2_MR13 : BOOL;
	{attribute addProperty Name "FSOE_Inp_D_2_MR14"}
	FSOE_Inp_D_2_MR14 : BOOL;
	{attribute addProperty Name "FSOE_Inp_D_2_MR15"}
	FSOE_Inp_D_2_MR15 : BOOL;
	{attribute addProperty Name "FSOE_Inp_D_2_MR16"}
	FSOE_Inp_D_2_MR16 : BOOL;
	{attribute addProperty Name "FSOE_Slave_CRC_2"}
	FSOE_Slave_CRC_2 : UINT;
	{attribute addProperty Name "FSOE_Inp_D_3_RES_49"}
	FSOE_Inp_D_3_RES_49 : BOOL;
	{attribute addProperty Name "FSOE_Inp_D_3_RES_50"}
	FSOE_Inp_D_3_RES_50 : BOOL;
	{attribute addProperty Name "FSOE_Inp_D_3_RES_51"}
	FSOE_Inp_D_3_RES_51 : BOOL;
	{attribute addProperty Name "FSOE_Inp_D_3_RES_52"}
	FSOE_Inp_D_3_RES_52 : BOOL;
	{attribute addProperty Name "FSOE_Inp_D_3_RES_53"}
	FSOE_Inp_D_3_RES_53 : BOOL;
	{attribute addProperty Name "FSOE_Inp_D_3_RES_54"}
	FSOE_Inp_D_3_RES_54 : BOOL;
	{attribute addProperty Name "FSOE_Inp_D_3_RES_55"}
	FSOE_Inp_D_3_RES_55 : BOOL;
	{attribute addProperty Name "FSOE_Inp_D_3_RES_56"}
	FSOE_Inp_D_3_RES_56 : BOOL;
	{attribute addProperty Name "FSOE_Inp_D_3_RES_57"}
	FSOE_Inp_D_3_RES_57 : BOOL;
	{attribute addProperty Name "FSOE_Inp_D_3_RES_58"}
	FSOE_Inp_D_3_RES_58 : BOOL;
	{attribute addProperty Name "FSOE_Inp_D_3_RES_59"}
	FSOE_Inp_D_3_RES_59 : BOOL;
	{attribute addProperty Name "FSOE_Inp_D_3_RES_60"}
	FSOE_Inp_D_3_RES_60 : BOOL;
	{attribute addProperty Name "FSOE_Inp_D_3_RES_61"}
	FSOE_Inp_D_3_RES_61 : BOOL;
	{attribute addProperty Name "FSOE_Inp_D_3_RES_62"}
	FSOE_Inp_D_3_RES_62 : BOOL;
	{attribute addProperty Name "FSOE_Inp_D_3_RES_63"}
	FSOE_Inp_D_3_RES_63 : BOOL;
	{attribute addProperty Name "FSOE_Inp_D_3_RES_64"}
	FSOE_Inp_D_3_RES_64 : BOOL;
	{attribute addProperty Name "FSOE_Slave_CRC_3"}
	FSOE_Slave_CRC_3 : UINT;
	{attribute addProperty Name "FSOE_ConnID"}
	FSOE_ConnID : UINT;
END_STRUCT
END_TYPE

// ---- DUTs/STRUCT/IO/PdoEntries/Status_F2CE6D91.TcDUT
{attribute 'GeneratedUsingTerminal: EL3024-0000-0019'}
{attribute addProperty BoxType "EL3024-0000-0019"}
{attribute addProperty Id "UnderrangeBOOL1OverrangeBOOL1Limit_1BYTE1Limit_2BYTE1ErrorBOOL1TxPDO_StateBOOL1TxPDO_ToggleBOOL1"}
{attribute addProperty CRC "4073614737"}
{attribute addProperty Size "7"}
TYPE Status_F2CE6D91 :
STRUCT
	{attribute addProperty Name "Underrange"}
	Underrange : BOOL;
	{attribute addProperty Name "Overrange"}
	Overrange : BOOL;
	{attribute addProperty Name "Limit_1"}
	Limit_1 : BYTE;
	{attribute addProperty Name "Limit_2"}
	Limit_2 : BYTE;
	{attribute addProperty Name "Error"}
	Error : BOOL;
	{attribute addProperty Name "TxPDO_State"}
	TxPDO_State : BOOL;
	{attribute addProperty Name "TxPDO_Toggle"}
	TxPDO_Toggle : BOOL;
END_STRUCT
END_TYPE

// ---- DUTs/STRUCT/IO/PDOs/AI_Standard_Channel_4A394481.TcDUT
{attribute 'GeneratedUsingTerminal: EL3024-0000-0019'}
{attribute addProperty BoxType "EL3024-0000-0019"}
{attribute addProperty Id "StatusAT %I*Status_F2CE6D917ValueAT %I*INT2"}
{attribute addProperty CRC "1245267073"}
{attribute addProperty Size "9"}
TYPE AI_Standard_Channel_4A394481 EXTENDS InputBase_8311D824 :
STRUCT
	{attribute addProperty Name "Status"}
	Status AT %I* : Status_F2CE6D91;
	{attribute addProperty Name "Value"}
	Value AT %I* : INT;
END_STRUCT
END_TYPE

// ---- DUTs/STRUCT/IO/PDOs/Channel_42CA91F7.TcDUT
{attribute 'GeneratedUsingTerminal: EL2634-0000-0017'}
{attribute addProperty BoxType "EL2634-0000-0017"}
{attribute addProperty Id "OutputAT %Q*BOOL1"}
{attribute addProperty CRC "1120571895"}
{attribute addProperty Size "1"}
TYPE Channel_42CA91F7 EXTENDS OutputBase_10CEE7DE :
STRUCT
	{attribute addProperty Name "Output"}
	Output AT %Q* : BOOL;
END_STRUCT
END_TYPE

// ---- DUTs/STRUCT/IO/PDOs/Compact_1DE69B90.TcDUT
{attribute 'GeneratedUsingTerminal: KRC4 secondary EL6695-1001-0004'}
{attribute addProperty BoxType "KRC4 secondary EL6695-1001-0004"}
{attribute addProperty Id "TxPDO_toggleAT %I*BOOL1TxPDO_stateAT %I*BOOL1External_device_not_connectedAT %I*BOOL1"}
{attribute addProperty CRC "501652368"}
{attribute addProperty Size "3"}
TYPE Compact_1DE69B90 EXTENDS InputBase_8311D824 :
STRUCT
	{attribute addProperty Name "TxPDO_toggle"}
	TxPDO_toggle AT %I* : BOOL;
	{attribute addProperty Name "TxPDO_state"}
	TxPDO_state AT %I* : BOOL;
	{attribute addProperty Name "External_device_not_connected"}
	External_device_not_connected AT %I* : BOOL;
END_STRUCT
END_TYPE

// ---- DUTs/STRUCT/IO/PDOs/InfoData_32EB74EA.TcDUT
{attribute 'GeneratedUsingTerminal: EL3024-0000-0019'}
{attribute addProperty BoxType "EL3024-0000-0019"}
{attribute addProperty Id "AdsAddrAT %I*AMSADDR8StateAT %I*UINT2"}
{attribute addProperty CRC "854291690"}
{attribute addProperty Size "10"}
TYPE InfoData_32EB74EA EXTENDS InputBase_8311D824 :
STRUCT
	{attribute addProperty Name "AdsAddr"}
	AdsAddr AT %I* : AMSADDR;
	{attribute addProperty Name "State"}
	State AT %I* : UINT;
END_STRUCT
END_TYPE

// ---- DUTs/STRUCT/IO/PDOs/InfoData_6F19DB2B.TcDUT
{attribute 'GeneratedUsingTerminal: EK1100-0000-0018'}
{attribute addProperty BoxType "EK1100-0000-0018"}
{attribute addProperty Id "StateAT %I*UINT2"}
{attribute addProperty CRC "1863965483"}
{attribute addProperty Size "2"}
TYPE InfoData_6F19DB2B :
STRUCT
	{attribute addProperty Name "State"}
	State AT %I* : UINT;
END_STRUCT
END_TYPE

// ---- DUTs/STRUCT/IO/PDOs/InfoData_8649EEEB.TcDUT
{attribute 'GeneratedUsingTerminal: IODEVICETYPE_ETHERCATPROT'}
{attribute addProperty BoxType "IODEVICETYPE_ETHERCATPROT"}
{attribute addProperty Id "ObjectIdAT %I*DWORD4StateAT %I*UINT2SlaveCountAT %I*UINT2"}
{attribute addProperty CRC "2252992235"}
{attribute addProperty Size "8"}
TYPE InfoData_8649EEEB EXTENDS InputBase_8311D824 :
STRUCT
	{attribute addProperty Name "ObjectId"}
	ObjectId AT %I* : DWORD;
	{attribute addProperty Name "State"}
	State AT %I* : UINT;
	{attribute addProperty Name "SlaveCount"}
	SlaveCount AT %I* : UINT;
END_STRUCT
END_TYPE

// ---- DUTs/STRUCT/IO/PDOs/InfoData_90184F0C.TcDUT
{attribute 'GeneratedUsingTerminal: KRC4 secondary EL6695-1001-0004'}
{attribute addProperty BoxType "KRC4 secondary EL6695-1001-0004"}
{attribute addProperty Id "AdsAddrAT %I*AMSADDR8AoeNetIdAT %I*AMSNETID6StateAT %I*UINT2"}
{attribute addProperty CRC "2417512204"}
{attribute addProperty Size "16"}
TYPE InfoData_90184F0C EXTENDS InputBase_8311D824 :
STRUCT
	{attribute addProperty Name "AdsAddr"}
	AdsAddr AT %I* : AMSADDR;
	{attribute addProperty Name "AoeNetId"}
	AoeNetId AT %I* : AMSNETID;
	{attribute addProperty Name "State"}
	State AT %I* : UINT;
END_STRUCT
END_TYPE

// ---- DUTs/STRUCT/IO/PDOs/InfoData_E68C61CD.TcDUT
{attribute 'GeneratedUsingTerminal: IODEVICETYPE_ETHERCATPROT'}
{attribute addProperty BoxType "IODEVICETYPE_ETHERCATPROT"}
{attribute addProperty Id "ChangeCountAT %I*UINT2DevIdAT %I*UINT2AmsNetIdAT %I*AMSNETID6CfgSlaveCountAT %I*UINT2DcToTcTimeOffsetAT %I*LINT8DcToExtTimeOffsetAT %I*LINT8"}
{attribute addProperty CRC "3867959757"}
{attribute addProperty Size "28"}
TYPE InfoData_E68C61CD EXTENDS InputBase_8311D824 :
STRUCT
	{attribute addProperty Name "ChangeCount"}
	ChangeCount AT %I* : UINT;
	{attribute addProperty Name "DevId"}
	DevId AT %I* : UINT;
	{attribute addProperty Name "AmsNetId"}
	AmsNetId AT %I* : AMSNETID;
	{attribute addProperty Name "CfgSlaveCount"}
	CfgSlaveCount AT %I* : UINT;
	{attribute addProperty Name "DcToTcTimeOffset"}
	DcToTcTimeOffset AT %I* : LINT;
	{attribute addProperty Name "DcToExtTimeOffset"}
	DcToExtTimeOffset AT %I* : LINT;
END_STRUCT
END_TYPE

// ---- DUTs/STRUCT/IO/PDOs/Inputs_A65FACA4.TcDUT
{attribute 'GeneratedUsingTerminal: IODEVICETYPE_ETHERCATPROT'}
{attribute addProperty BoxType "IODEVICETYPE_ETHERCATPROT"}
{attribute addProperty Id "SlaveCountAT %I*UINT2DevStateAT %I*UINT2Frm0StateAT %I*UINT2Frm0WcStateAT %I*UINT2Frm0InputToggleAT %I*UINT2"}
{attribute addProperty CRC "2791287972"}
{attribute addProperty Size "10"}
TYPE Inputs_A65FACA4 EXTENDS InputBase_8311D824 :
STRUCT
	{attribute addProperty Name "SlaveCount"}
	SlaveCount AT %I* : UINT;
	{attribute addProperty Name "DevState"}
	DevState AT %I* : UINT;
	{attribute addProperty Name "Frm0State"}
	Frm0State AT %I* : UINT;
	{attribute addProperty Name "Frm0WcState"}
	Frm0WcState AT %I* : UINT;
	{attribute addProperty Name "Frm0InputToggle"}
	Frm0InputToggle AT %I* : UINT;
END_STRUCT
END_TYPE

// ---- DUTs/STRUCT/IO/PDOs/Inputs_Bitf_43DA21F5.TcDUT
{attribute 'GeneratedUsingTerminal: KRC4 secondary EL6695-1001-0004'}
{attribute addProperty BoxType "KRC4 secondary EL6695-1001-0004"}
{attribute addProperty Id "FSOEAT %I*FSOE_892AE69275"}
{attribute addProperty CRC "1138369013"}
{attribute addProperty Size "75"}
TYPE Inputs_Bitf_43DA21F5 EXTENDS InputBase_8311D824 :
STRUCT
	{attribute addProperty Name "FSOE"}
	FSOE AT %I* : FSOE_892AE692;
END_STRUCT
END_TYPE

// ---- DUTs/STRUCT/IO/PDOs/Module_1_Sync_Inputs_26A07CFD.TcDUT
{attribute 'GeneratedUsingTerminal: KRC4 secondary EL6695-1001-0004'}
{attribute addProperty BoxType "KRC4 secondary EL6695-1001-0004"}
{attribute addProperty Id "CompactCompact_1DE69B903"}
{attribute addProperty CRC "648051965"}
{attribute addProperty Size "3"}
TYPE Module_1_Sync_Inputs_26A07CFD :
STRUCT
	{attribute addProperty Name "Compact"}
	Compact  : Compact_1DE69B90;
END_STRUCT
END_TYPE

// ---- DUTs/STRUCT/IO/PDOs/Module_2_Safety_Data_Bitf_8_Byte_x_D7FC8792.TcDUT
{attribute 'GeneratedUsingTerminal: KRC4 secondary EL6695-1001-0004'}
{attribute addProperty BoxType "KRC4 secondary EL6695-1001-0004"}
{attribute addProperty Id "Inputs_BitfInputs_Bitf_43DA21F575Outputs_BitfOutputs_Bitf_2744F33675"}
{attribute addProperty CRC "3623651218"}
{attribute addProperty Size "150"}
TYPE Module_2_Safety_Data_Bitf_8_Byte_x_D7FC8792 :
STRUCT
	{attribute addProperty Name "Inputs_Bitf"}
	Inputs_Bitf  : Inputs_Bitf_43DA21F5;
	{attribute addProperty Name "Outputs_Bitf"}
	Outputs_Bitf  : Outputs_Bitf_2744F336;
END_STRUCT
END_TYPE

// ---- DUTs/STRUCT/IO/PDOs/Module_3_Default_IO_1C907BA3.TcDUT
{attribute 'GeneratedUsingTerminal: KRC4 secondary EL6695-1001-0004'}
{attribute addProperty BoxType "KRC4 secondary EL6695-1001-0004"}
{attribute addProperty Id "Std_In_4_BytesStd_In_4_Bytes_89628F684Std_Out_4_BytesStd_Out_4_Bytes_1F5BD6B74"}
{attribute addProperty CRC "479230883"}
{attribute addProperty Size "8"}
TYPE Module_3_Default_IO_1C907BA3 :
STRUCT
	{attribute addProperty Name "Std_In_4_Bytes"}
	Std_In_4_Bytes  : Std_In_4_Bytes_89628F68;
	{attribute addProperty Name "Std_Out_4_Bytes"}
	Std_Out_4_Bytes  : Std_Out_4_Bytes_1F5BD6B7;
END_STRUCT
END_TYPE

// ---- DUTs/STRUCT/IO/PDOs/Outputs_23C0ED1D.TcDUT
{attribute 'GeneratedUsingTerminal: IODEVICETYPE_ETHERCATPROT'}
{attribute addProperty BoxType "IODEVICETYPE_ETHERCATPROT"}
{attribute addProperty Id "DevCtrlAT %Q*UINT2Frm0CtrlAT %Q*UINT2Frm0WcCtrlAT %Q*UINT2"}
{attribute addProperty CRC "599846173"}
{attribute addProperty Size "6"}
TYPE Outputs_23C0ED1D EXTENDS OutputBase_10CEE7DE :
STRUCT
	{attribute addProperty Name "DevCtrl"}
	DevCtrl AT %Q* : UINT;
	{attribute addProperty Name "Frm0Ctrl"}
	Frm0Ctrl AT %Q* : UINT;
	{attribute addProperty Name "Frm0WcCtrl"}
	Frm0WcCtrl AT %Q* : UINT;
END_STRUCT
END_TYPE

// ---- DUTs/STRUCT/IO/PDOs/Outputs_Bitf_2744F336.TcDUT
{attribute 'GeneratedUsingTerminal: KRC4 secondary EL6695-1001-0004'}
{attribute addProperty BoxType "KRC4 secondary EL6695-1001-0004"}
{attribute addProperty Id "FSOEAT %Q*FSOE_8292E3BB75"}
{attribute addProperty CRC "658830134"}
{attribute addProperty Size "75"}
TYPE Outputs_Bitf_2744F336 EXTENDS OutputBase_10CEE7DE :
STRUCT
	{attribute addProperty Name "FSOE"}
	FSOE AT %Q* : FSOE_8292E3BB;
END_STRUCT
END_TYPE

// ---- DUTs/STRUCT/IO/PDOs/Std_In_4_Bytes_89628F68.TcDUT
{attribute 'GeneratedUsingTerminal: KRC4 secondary EL6695-1001-0004'}
{attribute addProperty BoxType "KRC4 secondary EL6695-1001-0004"}
{attribute addProperty Id "Input_DWORD_0AT %I*UDINT4"}
{attribute addProperty CRC "2304937832"}
{attribute addProperty Size "4"}
TYPE Std_In_4_Bytes_89628F68 EXTENDS InputBase_8311D824 :
STRUCT
	{attribute addProperty Name "Input_DWORD_0"}
	Input_DWORD_0 AT %I* : UDINT;
END_STRUCT
END_TYPE

// ---- DUTs/STRUCT/IO/PDOs/Std_Out_4_Bytes_1F5BD6B7.TcDUT
{attribute 'GeneratedUsingTerminal: KRC4 secondary EL6695-1001-0004'}
{attribute addProperty BoxType "KRC4 secondary EL6695-1001-0004"}
{attribute addProperty Id "Output_DWORD_0AT %Q*UDINT4"}
{attribute addProperty CRC "526112439"}
{attribute addProperty Size "4"}
TYPE Std_Out_4_Bytes_1F5BD6B7 EXTENDS OutputBase_10CEE7DE :
STRUCT
	{attribute addProperty Name "Output_DWORD_0"}
	Output_DWORD_0 AT %Q* : UDINT;
END_STRUCT
END_TYPE

// ---- DUTs/STRUCT/IO/PDOs/WcState_0B2B16F9.TcDUT
{attribute 'GeneratedUsingTerminal: EL2634-0000-0017'}
{attribute addProperty BoxType "EL2634-0000-0017"}
{attribute addProperty Id "WcStateAT %I*BOOL1"}
{attribute addProperty CRC "187373305"}
{attribute addProperty Size "1"}
TYPE WcState_0B2B16F9 :
STRUCT
	{attribute addProperty Name "WcState"}
	WcState AT %I* : BOOL;
END_STRUCT
END_TYPE

// ---- DUTs/STRUCT/IO/PDOs/WcState_9091E0EB.TcDUT
{attribute 'GeneratedUsingTerminal: EL3024-0000-0019'}
{attribute addProperty BoxType "EL3024-0000-0019"}
{attribute addProperty Id "WcStateAT %I*BOOL1InputToggleAT %I*BOOL1"}
{attribute addProperty CRC "2425479403"}
{attribute addProperty Size "2"}
TYPE WcState_9091E0EB :
STRUCT
	{attribute addProperty Name "WcState"}
	WcState AT %I* : BOOL;
	{attribute addProperty Name "InputToggle"}
	InputToggle AT %I* : BOOL;
END_STRUCT
END_TYPE

// ---- DUTs/STRUCT/IO/Topology/E_Bus_F0495AE1.TcDUT
{attribute 'GeneratedUsingTerminal: IODEVICETYPE_ETHERCATPROT'}
{attribute addProperty BoxType "IODEVICETYPE_ETHERCATPROT"}
{attribute addProperty Id "Term_1_EK1100Term_1_EK1100_53501D3255X001_KRC4_secondary_EL6695_1001KRC4_secondary_EL6695_4F43E7C3179SyncUnitsSyncUnits_67D36DDA18InputsInputs_A65FACA410OutputsOutputs_23C0ED1D6InfoDataInfoData_E68C61CD28"}
{attribute addProperty CRC "4031339233"}
{attribute addProperty Size "296"}
{attribute addProperty Name "E-Bus"}
TYPE E_Bus_F0495AE1 EXTENDS EtcMasterBase_62654B43 :
STRUCT
	{attribute addProperty Name "Term 1 (EK1100)"}
	{attribute addProperty PreviousPort "E-Bus : Master"}
	{attribute addProperty SyncUnit "default"}
	Term_1_EK1100 : Term_1_EK1100_53501D32;
	{attribute addProperty Name "X001 (KRC4 secondary EL6695-1001)"}
	{attribute addProperty PreviousPort "Term 1 (EK1100) : C"}
	{attribute addProperty SyncUnit "default"}
	X001_KRC4_secondary_EL6695_1001 : KRC4_secondary_EL6695_4F43E7C3;
	{attribute addProperty Name "SyncUnits"}
	SyncUnits : SyncUnits_67D36DDA;
	{attribute addProperty Name "Inputs"}
	Inputs : Inputs_A65FACA4;
	{attribute addProperty Name "Outputs"}
	Outputs : Outputs_23C0ED1D;
	{attribute addProperty Name "InfoData"}
	InfoData : InfoData_E68C61CD;
END_STRUCT
END_TYPE

// ---- DUTs/STRUCT/IO/Topology/Term_1_EK1100_53501D32.TcDUT
{attribute 'GeneratedUsingTerminal: EK1100-0000-0018'}
{attribute addProperty BoxType "EK1100-0000-0018"}
{attribute addProperty Id "Term_2_EL3024EL3024_C4269E3248Term_3_EL2634EL2634_7B64371E7"}
{attribute addProperty CRC "1397759282"}
{attribute addProperty Size "55"}
{attribute addProperty Name "Term 1 (EK1100)"}
TYPE Term_1_EK1100_53501D32 EXTENDS EK1100_1FC0878B :
STRUCT
	{attribute addProperty Name "Term 2 (EL3024)"}
	{attribute addProperty PreviousPort "Term 1 (EK1100) : B"}
	{attribute addProperty SyncUnit "default"}
	Term_2_EL3024 : EL3024_C4269E32;
	{attribute addProperty Name "Term 3 (EL2634)"}
	{attribute addProperty PreviousPort "Term 2 (EL3024) : B"}
	{attribute addProperty SyncUnit "default"}
	Term_3_EL2634 : EL2634_7B64371E;
END_STRUCT
END_TYPE

// ---- GVLs/GVL_iXlinker.TcGVL
{attribute 'qualified_only'}
VAR_GLOBAL
		E_Bus : E_Bus_F0495AE1; // ONLY FB_Topology.E_Bus_Raw shall use this variable! iXlinker only generates Globals at the time of creating this project.
END_VAR

// ---- POUs/Cell/_Interface/I_HydrualicPump.TcIO
INTERFACE I_HydrualicPump

METHOD getSignal : BOOL
VAR_INPUT
END_VAR
END_METHOD

METHOD getState : eState
VAR_INPUT
END_VAR
END_METHOD

METHOD reset : BOOL
VAR_INPUT
END_VAR
END_METHOD

METHOD start : BOOL
VAR_INPUT
END_VAR
END_METHOD

METHOD stop : BOOL
VAR_INPUT
END_VAR
END_METHOD

END_INTERFACE

// ---- POUs/Cell/_Interface/I_PressureSensor.TcIO
INTERFACE I_PressureSensor

METHOD getSignal : LREAL
VAR_INPUT
END_VAR
END_METHOD

METHOD setSignal : BOOL
VAR_INPUT
    input : LREAL;
END_VAR
END_METHOD

END_INTERFACE

// ---- POUs/Cell/_Interface/I_Robot.TcIO
INTERFACE I_Robot

METHOD abort : BOOL
VAR_INPUT
END_VAR
END_METHOD

METHOD getState : eState
VAR_INPUT
END_VAR
END_METHOD

METHOD hold : BOOL
VAR_INPUT
END_VAR
END_METHOD

METHOD reset : BOOL
VAR_INPUT
END_VAR
END_METHOD

METHOD start : BOOL
VAR_INPUT
END_VAR
END_METHOD

METHOD stop : BOOL
VAR_INPUT
END_VAR
END_METHOD

END_INTERFACE

// ---- POUs/MAIN.TcPOU
PROGRAM MAIN
VAR
	//Config : ST_Configuration;
	VariantControl : FB_VariantControl;
	
	Cell : FB_Cell;
    HMI : FB_HMI;
END_VAR

// load machine config data
VariantControl(bLoadJSONFirstScan:=_TaskInfo[1].FirstCycle,
               bWriteJSON := HMI.HMItoPLC.variantControl.bExportJSON,
               Config := HMI.HMItoPLC.variantControl.Config);

// Don't execute anything until configuration data is loaded
IF VariantControl.bDone AND NOT VariantControl.bBusy THEN
    //Config := HMI.HMItoPLC.variantControl.Config;
    Cell(Config := HMI.HMItoPLC.variantControl.Config,
        HMItoPLC := HMI.HMItoPLC,
        PLCtoHMI => HMI.PLCtoHMI);

END_IF

// Run HMI as soon as machine config is loaded or failed to create config file
IF VariantControl.bDone THEN

    HMI.PLCtoHMI.variantControl.bNeedsCellDefinition := VariantControl.bLoadError;
    HMI();

END_IF

END_PROGRAM

// ---- POUs/FB_VariantControl.TcPOU
FUNCTION_BLOCK FB_VariantControl
VAR_IN_OUT
    Config : ST_Configuration;
END_VAR
VAR_INPUT
	bLoadJSONFirstScan : BOOL; // Executes on rising edge
    bWriteJSON : BOOL;
END_VAR
VAR_OUTPUT
	bDone : BOOL;
	bBusy : BOOL;
	
	//stConfigOut : ST_Configuration;
    bLoadError : BOOL;
END_VAR
VAR
	//JSON Settings handling variables
	bSaveJSON					: BOOL;
	bHasMember 					: BOOL;
	sCurrentMemberName 			: STRING;
	sJsonDoc       				: STRING(255);   
	sJsonDoc2      				: STRING(2000);   	
	sFilePath 					: STRING := 'C:\TwinCAT\MachineConfig.json';		
	
	rTrigSaveJSON 				: R_TRIG;
	fTrigLoadJSON 				: R_TRIG;
	
	//Variables for JSON handling
	fbJSONSaveLoad				: FB_JsonDomParser;
	fbJson         				: FB_JsonSaxWriter;  
	fbJsonDataType 				: FB_JsonReadWriteDataType;  
	fbJsonDOM 					: FB_JsonDomParser;
	jsonDoc 					: SJsonValue;
	jsonProp 					: SJsonValue;

	bLoadDone : BOOL;
	bLoadExecute : BOOL;
	bLoadJson : BOOL;
    
    bFoundSomething : BOOL;
    bFoundBoolValue : BOOL;
    bFoundStringValue : STRING;
END_VAR

rTrigSaveJSON(CLK := bWriteJSON); // to manually create file after changes or what not toggle this to export json file, don't forget to first toggle bits from stConfig!
IF rTrigSaveJSON.Q THEN
	
	bWriteJSON := FALSE;
	
	fbJson.ResetDocument();
	fbJsonDataType.AddJsonValueFromSymbol(fbJson, 'ST_Configuration', SIZEOF(Config), ADR(Config));
	sJsonDoc := fbJson.GetDocument();
	fbJson.CopyDocument(sJsonDoc2, SIZEOF(sJsonDoc2));
	fbJSONSaveLoad.ParseDocument(sJsonDoc2);

	bSaveJSON := TRUE;
	bLoadDone := TRUE;
	bLoadError := FALSE;
	
END_IF


IF fbJSONSaveLoad.SaveDocumentToFile(sFilePath, bSaveJSON) THEN
	bBusy := FALSE;
	bDone := TRUE;
END_IF


IF bLoadJSONFirstScan AND NOT bLoadExecute THEN
	bLoadExecute := bLoadJSONFirstScan;
	bBusy := TRUE;
END_IF


IF fbJSONSaveLoad.LoadDocumentFromFile(sFilePath, bLoadExecute) AND NOT bLoadDone THEN 
	bLoadDone:= TRUE;
	bLoadExecute := FALSE;
	bLoadJson := TRUE;
END_IF


IF NOT bLoadExecute AND NOT bLoadDone THEN
	bLoadError := TRUE;
    bDone := TRUE;
END_IF


fTrigLoadJSON(CLK := bLoadJson); //trigger for load file done
IF fTrigLoadJSON.Q THEN
	
    fbJSONSaveLoad.CopyDocument(sJsonDoc2, SIZEOF(sJsonDoc2));

    jsonDoc := fbJsonDOM.ParseDocument(sJsonDoc2);

    Config.sVersionHW := GetString('sVersionHW');
    Config.sVersionSW := GetString('sVersionSW');
    Config.bIsV1_0_0 := GetBool('bIsV1_0_0');
    Config.bIsSimulator := GetBool('bIsSimulator');

    // add as many as you desire below vvvvv
	
	bLoadJson := FALSE;
    bLoadError := FALSE;
	bDone := TRUE;
	bBusy := FALSE;
	
END_IF

METHOD GetBool : BOOL
VAR_INPUT
    memberName : STRING;
END_VAR
sCurrentMemberName := memberName;
bHasMember := fbJsonDOM.HasMember(jsonDoc, sCurrentMemberName);
IF (bHasMember) THEN
    bHasMember := FALSE;
    jsonProp := fbJsonDOM.FindMember(jsonDoc, sCurrentMemberName);
    GetBool := fbJsonDOM.GetBool(jsonProp);
ELSE
    GetBool := FALSE;
END_IF
END_METHOD

METHOD GetString : STRING
VAR_INPUT
    memberName : STRING;
END_VAR
sCurrentMemberName := memberName;
bHasMember := fbJsonDOM.HasMember(jsonDoc, sCurrentMemberName);
IF (bHasMember) THEN
    bHasMember := FALSE;
    jsonProp := fbJsonDOM.FindMember(jsonDoc, sCurrentMemberName);
    GetString := fbJsonDOM.GetString(jsonProp);
ELSE
    GetString := '';
END_IF
END_METHOD

END_FUNCTION_BLOCK

// ---- POUs/Cell/FB_Cell.TcPOU
FUNCTION_BLOCK FB_Cell
VAR_INPUT
	Config : ST_Configuration;
    HMItoPLC : st_HMItoPLC;
END_VAR
VAR_OUTPUT
	bBusy : BOOL;
    PLCtoHMI : st_PLCtoHMI;
END_VAR
VAR
	topology : FB_Topology;
	HydrualicsSystem : FB_HydrualicSystem;

    pretendFullFledgedScheduler : TON := (pt:=T#8S);
    
    // Robot
    fbFanucRobot : FB_Fanuc;
    fbKukaRobot_krc2 : FB_Kuka_KRC2;
    fbKukaRobot_krc4 : FB_Kuka_KRC4;
    fbRobotSim : FB_Robot_Simulator;
    iRobot : I_Robot;
    
    cellState : eCellState;
END_VAR

HandleInput();
VariantControl();

IF cellState <> eCellState.eCellState_Error THEN
	// cell logic
	IF NOT bBusy THEN
        IF HMItoPLC.cell.bGoToAuto THEN
			cellState := eCellState.eCellState_Automatic;
            PLCtoHMI.cell.bGoToAuto := NOT HMItoPLC.cell.bGoToAuto;
        ELSIF HMItoPLC.cell.bGoToManual THEN
			cellState := ecellstate.eCellState_Manual;
            PLCtoHMI.cell.bGoToManual := NOT HMItoPLC.cell.bGoToManual;
		END_IF
	END_IF

	// execute state methods
	IF cellState = eCellState.eCellState_Automatic THEN
		ExecuteAuto();
	ELSIF cellState = ecellstate.eCellState_Manual THEN
		ExecuteManual();
	END_IF
ELSE
    IF HMItoPLC.cell.bReset THEN
		ExecuteReset();
	END_IF
END_IF


pretendFullFledgedScheduler();
HydrualicsSystem();
fbFanucRobot();
fbKukaRobot_krc2();
fbKukaRobot_krc4();
fbRobotSim();

HandleOutput();

METHOD ExecuteAuto : BOOL
VAR_INPUT
END_VAR
IF NOT bBusy (*AND cellRobotManager.taskListEmpty()?*) THEN
    bBusy := TRUE;
END_IF

IF bBusy THEN

    IF cellState <> eCellState_Error THEN
        HydrualicsSystem.start();
    END_IF

    // start robot as soon as hydrualic system is ready
    IF HydrualicsSystem.getState() = eState_Running THEN
        IF pretendFullFledgedScheduler.Q THEN
            IF iRobot.getState() = eState_Idle THEN
                iRobot.start();
            END_IF
            pretendFullFledgedScheduler(IN := FALSE);
        ELSE
            // throw error
        END_IF
    END_IF

    IF iRobot.getState() = eState_Complete THEN
        IF NOT Config.bIsSimulator THEN
            bBusy := FALSE;
        END_IF
    ELSIF (iRobot.getState() = eState_Idle) AND HMItoPLC.cell.bGoToManual THEN
        // allow robot to complete current task and then go to manual
        bBusy := FALSE;
    ELSIF iRobot.getState() = eState_Error THEN
        // Throw cell into error state if there's a robot error
        cellState := eCellState_Error;
        bBusy := FALSE;
    END_IF
    
    IF HydrualicsSystem.getState() = eState_Error THEN
        cellState := eCellState_Error;
        iRobot.abort();
        bBusy := FALSE;
	END_IF
ELSE
    iRobot.stop();
    HydrualicsSystem.stop();
END_IF
END_METHOD

METHOD ExecuteManual : BOOL
VAR_INPUT
END_VAR
// not implemented

IF cellState = eCellState_Error THEN
    iRobot.hold();
END_IF

IF HydrualicsSystem.getState() = eState_Error THEN
    cellState := eCellState_Error;
END_IF

IF iRobot.getState() = eState_Error THEN
    cellState := eCellState_Error;
END_IF
END_METHOD

METHOD ExecuteReset : BOOL
VAR_INPUT
END_VAR


// reset alarms for cell and every subsystem and go to manual
cellState := eCellState_Manual;
iRobot.reset();
HydrualicsSystem.reset();
END_METHOD

METHOD HandleInput : BOOL
VAR_INPUT
END_VAR
topology.HandleInputs();

pretendFullFledgedScheduler.IN := TRUE;

fbKukaRobot_krc4.HardwareInputs.fault := topology.IOtoPLC.robot.fault;
fbRobotSim.HardwareInputs.fault := topology.IOtoPLC.robot.fault;
fbRobotSim.simCellState := cellState;
fbRobotSim.simHydroState := HydrualicsSystem.getState();


HydrualicsSystem.PressureSensor_input.value := topology.IOtoPLC.pressureTransducer.value;
HydrualicsSystem.bIsSimulator := Config.bIsSimulator;
HydrualicsSystem.bHasPump := Config.bHasPump;
HydrualicsSystem.sTypeOfPump := Config.sPumpType;
HydrualicsSystem.bHasPressureSensor := Config.bHasPressureSensor;
HydrualicsSystem.sTypeOfPressureSensor := Config.sPressureSensorType;
END_METHOD

METHOD HandleOutput : BOOL
VAR_INPUT
END_VAR
topology.PLCtoIO.robot.fault := fbKukaRobot_krc4.HardwareOutputs.fault OR fbRobotSim.HardwareOutputs.fault;

topology.PLCtoIO.hydroPump.On := HydrualicsSystem.hydrualicPump_output.On;

// send data to HMI struct
PLCtoHMI.cell.state := cellState;
PLCtoHMI.robot.state := iRobot.getState();
PLCtoHMI.hydrualics.state := HydrualicsSystem.PLCtoHMI.state;
PLCtoHMI.hydrualics.pump.state := HydrualicsSystem.PLCtoHMI.pump.state;
PLCtoHMI.hydrualics.psiSensor.value := HydrualicsSystem.PLCtoHMI.psiSensor.value;

PLCtoHMI.cell.bReset := HMItoPLC.cell.bReset;

topology.HandleOutputs();
END_METHOD

METHOD VariantControl : BOOL
VAR_INPUT
END_VAR
IF Config.bIsSimulator THEN
    iRobot := fbRobotSim;
ELSE
    // choose normal type according to MachineConfig.json file

    iRobot := fbKukaRobot_krc4;
END_IF
END_METHOD

END_FUNCTION_BLOCK

// ---- POUs/Cell/Hardware_IO/FB_Topology.TcPOU
FUNCTION_BLOCK FB_Topology
VAR_INPUT
    PLCtoIO : st_IO_Outputs; // hardware outputs
END_VAR
VAR_OUTPUT
	IOtoPLC : st_IO_Inputs; // hardware inputs
END_VAR
VAR
END_VAR

// monitor IO

METHOD HandleInputs : BOOL
VAR_INPUT
END_VAR
// ============ Hydrualic System ============

// Pressure Transducer
IOtoPLC.pressureTransducer.value := GVL_iXlinker.E_Bus.Term_1_EK1100.Term_2_EL3024.AI_Standard_Channel_1.Value;


// Proportional Valve


// Robot
IOtoPLC.robot.fault := GVL_iXlinker.E_Bus.X001_KRC4_secondary_EL6695_1001.Module_3_Default_IO.Std_In_4_Bytes.Input_DWORD_0.0;
END_METHOD

METHOD HandleOutputs : BOOL
VAR_INPUT
END_VAR
// Robot
GVL_iXlinker.E_Bus.X001_KRC4_secondary_EL6695_1001.Module_3_Default_IO.Std_Out_4_Bytes.Output_DWORD_0.0 := PLCtoIO.robot.fault;

// Pump
GVL_iXlinker.E_Bus.Term_1_EK1100.Term_3_EL2634.Channel_1.Output := PLCtoIO.hydroPump.On;
END_METHOD

END_FUNCTION_BLOCK

// ---- POUs/Cell/Hydrualics/FB_HydrualicSystem.TcPOU
FUNCTION_BLOCK FB_HydrualicSystem EXTENDS StateMachineBase
VAR_INPUT
    bIsSimulator : BOOL;

	// Hydrualic pump
	bHasPump : BOOL;
	sTypeOfPump : STRING;

	// Pressure sensor
	bHasPressureSensor : BOOL;
	sTypeOfPressureSensor : STRING;

    PressureSensor_input : st_PressureTransducer_Input;
END_VAR
VAR_OUTPUT
    bBusy : BOOL;
    bError : BOOL;
    bDone : BOOL;
    
    hydrualicPump_output : ST_Pump_Output;

    PLCtoHMI : st_PLCtoHMI_Hydrualics;
END_VAR
VAR
	// Function block instances for Hydrualic Pump
	fbPumpRealy : FB_Pump_RelayOnly;
	fbPumpHPU : FB_Pump_HPU;
    fbPumpSim : FB_Pump_Simulator;
    // Interface to pump
	iHydrualicPump : I_HydrualicPump;

    // Function block instances for Pressure Sensor
	fbPressureSensorSim : FB_PressureTransceiver_Sim;
	fbGenericPressureSensor : FB_GenericBrand_Transceiver;
    // Interface to Pressure Sensor
	iPressureSensor : I_PressureSensor;

    PressureValueMem : LREAL;

    primePumpTimeoutTON : TON := (PT := T#500ms);
    
END_VAR

M_VariantControl();
HandleInputs();

MonitorErrors();

ExecuteState();
IF NOT (nextState = curState) THEN
	StateTransition();
END_IF

fbPumpRealy();
fbPumpHPU();
fbPumpSim();
fbPressureSensorSim(simCellState := cellState);
fbGenericPressureSensor();

HandleOutputs();

ACTION ExecuteState:


CASE curState OF
	eState_Idle: ExecuteState_Idle();
	eState_Startup: ExecuteState_Startup();
	eState_Running: ExecuteState_Running();
	eState_Complete: ExecuteState_Complete();
	eState_Error: ExecuteState_Error();
	eState_Independent: ExecuteState_Independent();
END_CASE
END_ACTION

ACTION ExecuteState_Complete:

END_ACTION

ACTION ExecuteState_Error:

// stop pump in case of error
IF NOT (iHydrualicPump.getState() = eState_Idle) AND NOT (iHydrualicPump.getState() = eState_Error) THEN
    iHydrualicPump.stop();
END_IF
END_ACTION

ACTION ExecuteState_Idle:

END_ACTION

ACTION ExecuteState_Independent:

END_ACTION

ACTION ExecuteState_Running:
// I would setup every type of control loop here in a case statemant
// here I'm only using one (bang bang) as what is there to control with just ON/OFF

IF iPressureSensor.getSignal() > 10 THEN
    nextState := eState_Error;
    // throw overpressure error
    RETURN;
END_IF

// bang bang control
IF iPressureSensor.getSignal() > 9.9 THEN
    IF NOT (iHydrualicPump.getState() = eState_Idle) THEN
        // stop once pressure is above set point
        iHydrualicPump.stop();
    END_IF
ELSIF iPressureSensor.getSignal() <= 8.2 THEN
    IF NOT (iHydrualicPump.getState() = eState_Running) THEN
        // start once pressure below minimun
        iHydrualicPump.start();
    END_IF
END_IF
END_ACTION

ACTION ExecuteState_Startup:

IF (iHydrualicPump.getState() = eState_Idle) AND NOT (iHydrualicPump.getState() = eState_Error) THEN
    iHydrualicPump.start();
ELSE
    // failed to start error
END_IF

IF iPressureSensor.getSignal() > 8 THEN
    nextState := eState_Running;
END_IF

primePumpTimeoutTON(IN := (PressureValueMem > iPressureSensor.getSignal()));
IF primePumpTimeoutTON.Q THEN
    // failed to pressureize system. Checks for leaks! Or faulty motor.
    nextState := eState_Error;
END_IF

IF iPressureSensor.getSignal() > PressureValueMem THEN
    PressureValueMem := iPressureSensor.getSignal();
END_IF
END_ACTION

METHOD HandleInputs : BOOL
VAR_INPUT
END_VAR

// Pass pressure value to iPressureSensor
IF bIsSimulator THEN
    // pass pump state back to pressure sensor to generate sim signal
    fbPressureSensorSim.bPumpIsON := iHydrualicPump.getState() = eState_Running;
ELSE
    iPressureSensor.setSignal(PressureSensor_input.value);    
END_IF
END_METHOD

METHOD HandleOutputs : BOOL
VAR_INPUT
END_VAR
// Set Outputs
hydrualicPump_output.On := iHydrualicPump.getSignal();

// populate HMI struct
PLCtoHMI.state := curState;
PLCtoHMI.psiSensor.value := iPressureSensor.getSignal();
PLCtoHMI.pump.state := iHydrualicPump.getState();
END_METHOD

METHOD PRIVATE M_VariantControl : BOOL
VAR_INPUT
END_VAR
// Handle hydrualic pump options
IF bIsSimulator THEN
    iHydrualicPump := fbPumpSim;
    iPressureSensor := fbPressureSensorSim;
ELSE
    IF sTypeOfPump='relay' THEN
        iHydrualicPump := fbPumpRealy;
    ELSIF sTypeOfPump='hpu' THEN
        iHydrualicPump := fbPumpHPU;
    ELSE
        iHydrualicPump := fbPumpRealy;
    END_IF
    
    iPressureSensor := fbGenericPressureSensor;
END_IF
END_METHOD

METHOD MonitorErrors : BOOL
VAR_INPUT
END_VAR
// error if hydrualic pump fails
IF iHydrualicPump.getState() = eState_Error THEN
    nextState := eState_Error;
    // throw pump error
END_IF

IF curState = eState_Running THEN
    IF iPressureSensor.getSignal() < 8 THEN
        iHydrualicPump.stop();
        nextState := eState_Error;
        // throw pressure drop error
    END_IF
END_IF
END_METHOD

METHOD reset : BOOL
resetAlarms();

iHydrualicPump.reset();

nextState := eState_Idle;
END_METHOD

METHOD start: BOOL
VAR_INPUT
END_VAR
IF curState = eState_Idle THEN
	nextState := eState_Startup;
	start := TRUE;
ELSE
	start := FALSE;
END_IF
END_METHOD

ACTION StateTransition:
//reset timers


IF nextState = eState_Startup THEN
	primePumpTimeoutTON(IN := FALSE);
    PressureValueMem := iPressureSensor.getSignal();
END_IF


SUPER^.StateTransition();
END_ACTION

END_FUNCTION_BLOCK

// ---- POUs/Cell/BaseClasses/StateMachineBase.TcPOU
FUNCTION_BLOCK StateMachineBase //IMPLEMENTS  iStateMachine
VAR_INPUT
	resourceID:INT;
END_VAR
VAR_OUTPUT
	//Current alarm code
		//Alarms
	Alarms: ARRAY [0..10] OF BOOL;
	InfoMsg: STRING;
END_VAR
VAR
	//State Machine
	prevState : eState;
	curState : eState;
	nextState : eState;
    HMIState : INT;
	
	cellState : eCellState;
    sTmpState : STRING(255);
    arrStateHistory : ARRAY [ 0..50 ] OF STRING(255);
END_VAR

METHOD abort : BOOL
VAR_INPUT
END_VAR
END_METHOD

METHOD getID : INT
getID:=resourceID;
END_METHOD

METHOD getState : eState
getState:=curState;
END_METHOD

METHOD hold : BOOL
hold := FALSE;
END_METHOD

METHOD ready : BOOL
VAR_INPUT
END_VAR
ready := TRUE;
END_METHOD

METHOD reset : BOOL
reset := FALSE;
END_METHOD

METHOD resetAlarms
VAR_INPUT
END_VAR
VAR
	i:INT;
	ToolData: INT;
END_VAR
FOR i:=1 TO 20 DO
	Alarms[i] := FALSE;
END_FOR
END_METHOD

METHOD resetInfoMsg
VAR_INPUT
END_VAR
InfoMsg := '';
END_METHOD

METHOD restart : BOOL
restart := FALSE;
END_METHOD

METHOD start : BOOL
start := FALSE;
END_METHOD

ACTION StateTransition:
IF curState = eState_error THEN
	resetAlarms();
END_IF

prevState := curState;
curState := nextState;
HMIState := CurState;


sTmpState := TO_STRING(nextState);
Queue_FIFO(
    inputSize   := SIZEOF(sTmpState),
    inputAdr    := ADR(sTmpState),
    arrSize := SIZEOF(arrStateHistory),
    arrAdr  := ADR(arrStateHistory)
);
END_ACTION

METHOD stop : BOOL
stop := FALSE;
END_METHOD

METHOD trackStateChange
VAR_INPUT
END_VAR
END_METHOD

END_FUNCTION_BLOCK

// ---- POUs/Functions/Queue_FIFO.TcPOU
FUNCTION Queue_FIFO : BOOL
VAR_INPUT
	inputSize : UDINT;
	inputAdr : POINTER TO BYTE;
	
	arrSize : UDINT;
	arrAdr : POINTER TO BYTE;
END_VAR
VAR
END_VAR

FW_MemMove(pDest := arrAdr + inputSize, pSrc := arrAdr, cbLen := arrSize - inputSize);

FW_MemMove(pDest := arrAdr, pSrc := inputAdr, cbLen := inputSize);

END_FUNCTION

// ---- POUs/Cell/Hydrualics/Pump/Types/FB_Pump_RelayOnly.TcPOU
FUNCTION_BLOCK FB_Pump_RelayOnly EXTENDS FB_Pump
VAR_INPUT
END_VAR
VAR_OUTPUT
    hydrualicPump_output : ST_Pump_Output;
END_VAR
VAR
END_VAR

ACTION ExecuteState:


CASE curState OF
	eState_Idle: ExecuteState_Idle();
	eState_Startup: ExecuteState_Startup();
	eState_Running: ExecuteState_Running();
	eState_Complete: ExecuteState_Complete();
    eState_Stopping: ExecuteState_Stopping();
    eState_Stopped: ExecuteState_Stopped();
	eState_Error: ExecuteState_Error();
	eState_Independent: ExecuteState_Independent();
END_CASE
END_ACTION

ACTION ExecuteState_Complete:

END_ACTION

ACTION ExecuteState_Error:
// Set Outputs
hydrualicPump_output.On := FALSE;
END_ACTION

ACTION ExecuteState_Idle:
// Set Outputs
hydrualicPump_output.On := FALSE;
END_ACTION

ACTION ExecuteState_Independent:
// Set Outputs
hydrualicPump_output.On := FALSE;
END_ACTION

ACTION ExecuteState_Running:
// Set Outputs
hydrualicPump_output.On := TRUE;
END_ACTION

ACTION ExecuteState_Startup:

// reset timers

// set output to true
nextState := eState_Running;
END_ACTION

ACTION ExecuteState_Stopped:
nextState := eState_Idle;
END_ACTION

ACTION ExecuteState_Stopping:
nextState := eState_Stopped;
END_ACTION

METHOD getSignal : BOOL
VAR_INPUT
END_VAR
getSignal := hydrualicPump_output.On;
END_METHOD

METHOD reset : BOOL
resetAlarms();

IF curState = eState_Complete THEN
	nextState := eState_Idle;
	reset := TRUE;
ELSIF curState = eState_Error THEN
    nextState := eState_Idle;
ELSE
	reset := FALSE;
END_IF
END_METHOD

METHOD start: BOOL
VAR_INPUT
END_VAR
IF curState = eState_Idle THEN
	nextState := eState_Startup;
	start := TRUE;
ELSE
	start := FALSE;
END_IF
END_METHOD

ACTION StateTransition:
SUPER^.StateTransition();
END_ACTION

END_FUNCTION_BLOCK

// ---- POUs/Cell/Hydrualics/Pump/FB_Pump.TcPOU
FUNCTION_BLOCK FB_Pump EXTENDS StateMachineBase IMPLEMENTS I_HydrualicPump
VAR_INPUT
    bIsSimulator : BOOL;
	bPumpRelay : BOOL; // Option: has pump with relay only
	bPumpHPU : BOOL; // Option: has Hydrualic Power Unit (HPU)
END_VAR
VAR_OUTPUT
END_VAR
VAR
    //fInputSignal : LREAL;
END_VAR

METHOD getSignal : BOOL
VAR_INPUT
END_VAR
END_METHOD

METHOD start : BOOL
VAR_INPUT
END_VAR
nextState := eState_Startup;
END_METHOD

METHOD stop : BOOL
VAR_INPUT
END_VAR
nextState := eState_Stopping;
END_METHOD

END_FUNCTION_BLOCK

// ---- POUs/Cell/Hydrualics/Pump/Types/FB_Pump_HPU.TcPOU
FUNCTION_BLOCK FB_Pump_HPU EXTENDS FB_Pump
VAR_INPUT
END_VAR
VAR_OUTPUT
END_VAR
VAR
END_VAR

// something fancy like this: https://whyps.com/basics-of-hydraulic-power-units

END_FUNCTION_BLOCK

// ---- POUs/Cell/Hydrualics/Pump/Types/FB_Pump_Simulator.TcPOU
FUNCTION_BLOCK FB_Pump_Simulator EXTENDS FB_Pump
VAR_INPUT
END_VAR
VAR_OUTPUT
    hydrualicPump_output : ST_Pump_Output;
END_VAR
VAR
END_VAR



ExecuteState();
IF NOT (nextState = curState)THEN
    StateTransition();
END_IF

ACTION ExecuteState:


CASE curState OF
	eState_Idle: ExecuteState_Idle();
	eState_Startup: ExecuteState_Startup();
	eState_Running: ExecuteState_Running();
	eState_Complete: ExecuteState_Complete();
    eState_Stopping: ExecuteState_Stopping();
    eState_Stopped: ExecuteState_Stopped();
	eState_Error: ExecuteState_Error();
	eState_Independent: ExecuteState_Independent();
END_CASE
END_ACTION

ACTION ExecuteState_Complete:

END_ACTION

ACTION ExecuteState_Error:
// Set Outputs
hydrualicPump_output.On := FALSE;
END_ACTION

ACTION ExecuteState_Idle:
// Set Outputs
hydrualicPump_output.On := FALSE;
END_ACTION

ACTION ExecuteState_Independent:
// Set Outputs
hydrualicPump_output.On := FALSE;
END_ACTION

ACTION ExecuteState_Running:
// Set Outputs
hydrualicPump_output.On := TRUE;
END_ACTION

ACTION ExecuteState_Startup:

// reset timers

// set output to true
nextState := eState_Running;
END_ACTION

ACTION ExecuteState_Stopped:
nextState := eState_Idle;
END_ACTION

ACTION ExecuteState_Stopping:
nextState := eState_Stopped;
END_ACTION

METHOD reset : BOOL
resetAlarms();

IF curState = eState_Complete THEN
	nextState := eState_Idle;
	reset := TRUE;
ELSIF curState = eState_Error THEN
    nextState := eState_Idle;
ELSE
	reset := FALSE;
END_IF
END_METHOD

METHOD start: BOOL
VAR_INPUT
END_VAR
IF curState = eState_Idle THEN
	nextState := eState_Startup;
	start := TRUE;
ELSE
	start := FALSE;
END_IF
END_METHOD

ACTION StateTransition:
SUPER^.StateTransition();
END_ACTION

END_FUNCTION_BLOCK

// ---- POUs/Cell/Hydrualics/PressureSensor/Types/FB_PressureTransceiver_Sim.TcPOU
FUNCTION_BLOCK FB_PressureTransceiver_Sim EXTENDS FB_PressureSensor
VAR_INPUT
    bPumpIsON : BOOL; // generates signal based on pump input
    simCellState : eCellState;
END_VAR
VAR_OUTPUT
END_VAR
VAR
    signalClimbTON : TON := (PT := T#25MS);
    signalFallTON : TON := (PT := T#50ms);
    
    simPressureDropTON : TON := (PT := T#70S);
END_VAR

IF bPumpIsON AND (curState = eState_Idle) THEN
    // simulate a rising signal when pump is ON
    nextState := eState_Startup;
END_IF

ExecuteState();
IF NOT (nextState = curState)THEN
    StateTransition();
END_IF

ACTION ExecuteState:


CASE curState OF
	eState_Idle: ExecuteState_Idle();
	eState_Startup: ExecuteState_Startup();
	eState_Running: ExecuteState_Running();
	eState_Complete: ExecuteState_Complete();
	eState_Error: ExecuteState_Error();
	eState_Independent: ExecuteState_Independent();
END_CASE
END_ACTION

ACTION ExecuteState_Complete:

END_ACTION

ACTION ExecuteState_Error:

END_ACTION

ACTION ExecuteState_Idle:

END_ACTION

ACTION ExecuteState_Independent:

END_ACTION

ACTION ExecuteState_Running:
IF bPumpIsON THEN

    // psi climbs
    signalClimbTON(IN := TRUE);
    IF signalClimbTON.Q THEN
        fBufferedSignal := fBufferedSignal + 0.1;
        signalClimbTON(IN := FALSE);
    END_IF

ELSE

    // psi falls
    IF fBufferedSignal < 2 THEN // if somehow signal falls below
        fBufferedSignal := 2;
    END_IF
    IF fBufferedSignal > 2 THEN // only if signal is more than hardware min decrease it
        signalFallTON(IN := TRUE);
        IF signalFallTON.Q THEN
            fBufferedSignal := fBufferedSignal - 0.01;
            signalFallTON(IN := FALSE);
        END_IF
	END_IF

END_IF


// every nth seconds simulate a pressure drop error
IF simCellState = eCellState_Automatic OR simCellState = eCellState_Manual THEN
    simPressureDropTON(IN := TRUE);
    IF simPressureDropTON.Q THEN
        fBufferedSignal := 2;
        simPressureDropTON(IN := FALSE);
    END_IF
END_IF
END_ACTION

ACTION ExecuteState_Startup:
// Build up pressure first

nextState := eState_Running;
END_ACTION

METHOD getSignal : LREAL
VAR_INPUT
END_VAR
// return signal value to outside world
getSignal := fBufferedSignal;
END_METHOD

METHOD setSignal : BOOL
VAR_INPUT
    input : LREAL;
END_VAR
fInputSignal := input;
END_METHOD

ACTION StateTransition:
//reset timers

SUPER^.StateTransition();
END_ACTION

END_FUNCTION_BLOCK

// ---- POUs/Cell/Hydrualics/PressureSensor/FB_PressureSensor.TcPOU
FUNCTION_BLOCK FB_PressureSensor EXTENDS StateMachineBase IMPLEMENTS I_PressureSensor
VAR_INPUT
    bIsSimulator : BOOL;
END_VAR
VAR_OUTPUT
END_VAR
VAR
    fInputSignal : LREAL; // 0-10v
    fBufferedSignal : LREAL; // 0-10v
END_VAR

METHOD getSignal : LREAL
VAR_INPUT
END_VAR
getSignal := 0;
END_METHOD

METHOD setSignal : BOOL
VAR_INPUT
    input : LREAL;
END_VAR
fInputSignal := input;
END_METHOD

END_FUNCTION_BLOCK

// ---- POUs/Cell/Hydrualics/PressureSensor/Types/FB_GenericBrand_Transceiver.TcPOU
FUNCTION_BLOCK FB_GenericBrand_Transceiver EXTENDS FB_PressureSensor
VAR_INPUT
END_VAR
VAR_OUTPUT
END_VAR
VAR
END_VAR

METHOD getSignal : LREAL
VAR_INPUT
END_VAR
// Pressure Transducer
 // Using 4..20mA input card with a 0-10v sensor. To make this possible a 500ohm resister was added. Best to buy the correct hardware.
 // Scale 4.20mA value to 2v-10v
fBufferedSignal := Scale(signal := fInputSignal,
                           inputMin := 0.0, // 4mA
                           inputMax := 32767.0, // 20mA
                           outputMin := 2, // 2v at 4mA
                           outputMax := 10);

getSignal := fBufferedSignal;
END_METHOD

METHOD setSignal : BOOL
VAR_INPUT
    input : LREAL;
END_VAR
fInputSignal := input;
END_METHOD

END_FUNCTION_BLOCK

// ---- POUs/Functions/Scale.TcPOU
FUNCTION Scale : LREAL
VAR_INPUT
	signal : LREAL;
	inputMin : LREAL;
	inputMax : LREAL;
	outputMin : LREAL;
	outputMax : LREAL;
END_VAR
VAR
END_VAR

IF signal < inputMin OR signal > inputMax THEN
	Scale := 0;
ELSE
	IF ((inputMax - inputMin) + outputMin) <> 0 THEN
	    Scale := ((signal - inputMin) * (outputMax - outputMin) / (inputMax - inputMin) + outputMin);
	ELSE
		Scale := 0;
	END_IF
END_IF

END_FUNCTION

// ---- POUs/Cell/Robots/6_axis/Types/FB_Fanuc.TcPOU
FUNCTION_BLOCK FB_Fanuc
VAR_INPUT
END_VAR
VAR_OUTPUT
END_VAR
VAR
END_VAR

END_FUNCTION_BLOCK

// ---- POUs/Cell/Robots/6_axis/Types/FB_Kuka_KRC2.TcPOU
FUNCTION_BLOCK FB_Kuka_KRC2
VAR_INPUT
END_VAR
VAR_OUTPUT
END_VAR
VAR
END_VAR

END_FUNCTION_BLOCK

// ---- POUs/Cell/Robots/6_axis/Types/FB_Kuka_KRC4.TcPOU
FUNCTION_BLOCK FB_Kuka_KRC4 EXTENDS FB_Robot
VAR_INPUT
    HardwareInputs : st_Robot_Input;
END_VAR
VAR_OUTPUT
    HardwareOutputs : st_Robot_Output;
END_VAR
VAR    
    StartupTimeoutTON : TON := (PT:=T#7S);
END_VAR



ExecuteState();
IF NOT (nextState = curState) THEN
	StateTransition();
END_IF;

ACTION ExecuteState:
// Watch for safety inputs from robot, e-stops, etc. and immediately goto state error
// IF RobotSafetyInput THEN
//  curState := eState_Error;
// END_IF


CASE curState OF
	eState_Idle: ExecuteState_Idle();
	eState_Startup: ExecuteState_Startup();
	eState_Running: ExecuteState_Running();
	eState_Complete: ExecuteState_Complete();
	eState_Error: ExecuteState_Error();
	eState_Independent: ExecuteState_Independent();
END_CASE
END_ACTION

ACTION ExecuteState_Complete:
//Output signals

nextState := eState_Idle;
END_ACTION

ACTION ExecuteState_Error:
//Output signals
HardwareOutputs.fault := TRUE;
END_ACTION

ACTION ExecuteState_Held:
//Set outputs
END_ACTION

ACTION ExecuteState_Holding:
//Set outputs

//Wait for held signal, then go to Held state
nextState := eState_Held;
END_ACTION

ACTION ExecuteState_Idle:
// monitor IO while idle
// set IO while in idle state

//Output signals
HardwareOutputs.fault := FALSE;
END_ACTION

ACTION ExecuteState_Independent:
//Output signals
END_ACTION

ACTION ExecuteState_Running:
//Output signals
END_ACTION

ACTION ExecuteState_Startup:
nextState := eState_Running;
END_ACTION

METHOD hold : BOOL
IF curState = eState_Running THEN
	nextState := eState_Holding;
	hold := TRUE;
ELSE
	hold := FALSE;
END_IF
END_METHOD

METHOD reset : BOOL
resetAlarms();

IF curState = eState_Complete THEN
	nextState := eState_Idle;
	reset := TRUE;
ELSIF curState = eState_Error THEN
	nextState := eState_Idle;
	reset := TRUE;
ELSE
	reset := FALSE;
END_IF
END_METHOD

METHOD start: BOOL
VAR_INPUT
END_VAR
IF curState = eState_Idle THEN
	nextState := eState_Startup;
	start := TRUE;
ELSE
	start := FALSE;
END_IF
END_METHOD

ACTION StateTransition:
//reset timers watchdog timers

SUPER^.StateTransition();
END_ACTION

END_FUNCTION_BLOCK

// ---- POUs/Cell/Robots/FB_Robot.TcPOU
FUNCTION_BLOCK FB_Robot EXTENDS StateMachineBase IMPLEMENTS I_Robot
VAR_INPUT
    bIsSimulator : BOOL;
END_VAR
VAR_OUTPUT
END_VAR
VAR
END_VAR

END_FUNCTION_BLOCK

// ---- POUs/Cell/Robots/6_axis/Types/FB_Robot_Simulator.TcPOU
FUNCTION_BLOCK FB_Robot_Simulator EXTENDS FB_Robot
VAR_INPUT
    simCellState : eCellState;
    simHydroState : eState;
    HardwareInputs : st_Robot_Input;
END_VAR
VAR_OUTPUT
    HardwareOutputs : st_Robot_Output;
END_VAR
VAR
    simRunningTON : TON := (PT:=T#10S);

    StartupTimeoutTON : TON := (PT:=T#7S);
END_VAR



ExecuteState();
IF NOT (nextState = curState) THEN
	StateTransition();
END_IF;

METHOD abort: BOOL;
VAR_INPUT
END_VAR
IF curState = eState_Running THEN
	nextState := eState_Error;
	abort := TRUE;
ELSE
	abort := FALSE;
END_IF
END_METHOD

ACTION ExecuteState:
// Watch for safety inputs and immediately goto state error
// IF SomeError THEN
//  curState := eState_Error;
// END_IF

CASE curState OF
	eState_Idle: ExecuteState_Idle();
	eState_Startup: ExecuteState_Startup();
	eState_Running: ExecuteState_Running();
    eState_Holding: ExecuteState_Holding();
    eState_Held: ExecuteState_Held();
	eState_Complete: ExecuteState_Complete();
	eState_Error: ExecuteState_Error();
	eState_Independent: ExecuteState_Independent();
END_CASE
END_ACTION

ACTION ExecuteState_Complete:
//Output signals

nextState := eState_Idle;
END_ACTION

ACTION ExecuteState_Error:
//Output signals
HardwareOutputs.fault := TRUE;
END_ACTION

ACTION ExecuteState_Held:
//Set outputs

IF simCellState = eCellState_Error THEN
    // in sim just put it back in idle
    nextState := eState_Idle;
END_IF
END_ACTION

ACTION ExecuteState_Holding:
//Set outputs

//Wait for held signal, then go to Held state
nextState := eState_Held;
END_ACTION

ACTION ExecuteState_Idle:
// monitor IO while idle
// set IO while in idle state

//Output signals
HardwareOutputs.fault := FALSE;
END_ACTION

ACTION ExecuteState_Independent:
//Output signals
END_ACTION

ACTION ExecuteState_Running:


simRunningTON(IN:=TRUE);
IF simRunningTON.Q THEN
    //simRaiseError_counter := simRaiseError_counter+1;
    nextState := eState_Complete;
END_IF

// error robot after nth cycle
//IF simRaiseError_counter = 5 THEN
//    nextState := eState_Error;
//    simRaiseError_counter := 0;
//END_IF
END_ACTION

ACTION ExecuteState_Startup:

nextState := eState_Running;
END_ACTION

METHOD hold : BOOL
IF curState = eState_Running THEN
	nextState := eState_Holding;
	hold := TRUE;
ELSE
	hold := FALSE;
END_IF
END_METHOD

METHOD reset : BOOL
resetAlarms();

IF curState = eState_Complete THEN
	nextState := eState_Idle;
	reset := TRUE;
ELSIF curState = eState_Error THEN // AND InputSignals.AutoMode AND InputSignals.Homed AND InputSignals.LoadUnloadReady AND NOT InputSignals.InCycle THEN
	nextState := eState_Idle;
	reset := TRUE;
ELSE
	reset := FALSE;
END_IF
END_METHOD

METHOD start: BOOL
VAR_INPUT
END_VAR
IF curState = eState_Idle THEN
	nextState := eState_Startup;
	start := TRUE;
ELSE
	start := FALSE;
END_IF
END_METHOD

ACTION StateTransition:
//reset timers watchdog timers

simRunningTON(in := FALSE);
StartupTimeoutTON(IN := FALSE);

IF nextState = eState_Startup THEN
	StartupTimeoutTON(IN := FALSE);
END_IF

IF nextState = eState_Startup THEN
	simRunningTON(IN := FALSE);
END_IF

SUPER^.StateTransition();
END_ACTION

END_FUNCTION_BLOCK

// ---- POUs/HMI/FB_HMI.TcPOU
FUNCTION_BLOCK FB_HMI
VAR_INPUT
    PLCtoHMI : st_PLCtoHMI;
END_VAR
VAR_OUTPUT
    HMItoPLC : st_HMItoPLC;
END_VAR
VAR
    delayWriteTON : TON := (PT := T#500MS);
    writeDurationTON : TON := (PT := T#50MS);
    //writeJson : BOOL;
END_VAR

IF PLCtoHMI.cell.state = eCellState_Error THEN
    HMItoPLC.hmi.bShowResetBtn := TRUE;
END_IF

IF HMItoPLC.cell.bReset THEN
    HMItoPLC.hmi.bShowResetBtn := FALSE;
END_IF

IF HMItoPLC.cell.bGoToAuto OR HMItoPLC.cell.bGoToManual THEN
    IF PLCtoHMI.cell.state = eCellState_Automatic THEN
        HMItoPLC.cell.bGoToAuto := FALSE;
    END_IF
    IF PLCtoHMI.cell.state = eCellState_Manual THEN
        HMItoPLC.cell.bGoToManual := FALSE;
    END_IF
END_IF

IF PLCtoHMI.variantControl.bNeedsCellDefinition THEN
    IF HMItoPLC.variantControl.bWriteJSON THEN
         delayWriteTON(IN := TRUE);
        IF delayWriteTON.Q THEN
            HMItoPLC.variantControl.bExportJSON := TRUE;
            HMItoPLC.variantControl.bWriteJSON := FALSE;
            delayWriteTON(IN := FALSE);
            writeDurationTON.IN := TRUE;
        END_IF
    END_IF
END_IF

writeDurationTON();
IF writeDurationTON.Q THEN
    HMItoPLC.variantControl.bExportJSON := FALSE;
    writeDurationTON.IN := FALSE;
END_IF

END_FUNCTION_BLOCK

// ---- POUs/Cell/Robots/Gantry/Types/FB_SomeGrantryRobot.TcPOU
FUNCTION_BLOCK FB_SomeGrantryRobot
VAR_INPUT
END_VAR
VAR_OUTPUT
END_VAR
VAR
END_VAR

END_FUNCTION_BLOCK
